LIN {X 0,Y 514.688,Z 526.81,A -85,B 0,C 180,E1 4924.755,E2 4924.755} C_VEL
LIN {X 0,Y 514.758,Z 527.266,A -85,B 0,C 180,E1 4925.27,E2 4925.27} C_VEL
LIN {X 0,Y 521.785,Z 550.887,A -85,B 0,C 180,E1 4925.881,E2 4925.881} C_VEL
LIN {X 0,Y 521.448,Z 608.09,A -85,B 0,C 180,E1 4926.837,E2 4926.837} C_VEL
LIN {X 0,Y 520.391,Z 641.868,A -85,B 0,C 180,E1 4928.058,E2 4928.058} C_VEL
LIN {X 0,Y 519.091,Z 674.479,A -85,B 0,C 180,E1 4929.962,E2 4929.962} C_VEL
LIN {X 0,Y 517.777,Z 702.458,A -85,B 0,C 180,E1 4932.319,E2 4932.319} C_VEL
LIN {X 0,Y 516.718,Z 728.108,A -85,B 0,C 180,E1 4935.321,E2 4935.321} C_VEL
LIN {X 0,Y 516.002,Z 747.013,A -85,B 0,C 180,E1 4938.414,E2 4938.414} C_VEL
LIN {X 0,Y 515.59,Z 761.456,A -85,B 0,C 180,E1 4941.986,E2 4941.986} C_VEL
LIN {X 0,Y 515.379,Z 770.612,A -85,B 0,C 180,E1 4945.792,E2 4945.792} C_VEL
LIN {X 0,Y 515.287,Z 773.417,A -85,B 0,C 180,E1 4948.32,E2 4948.32} C_VEL
LIN {X 0,Y 515.26,Z 773.413,A -85,B 0,C 180,E1 4951.688,E2 4951.688} C_VEL
LIN {X 0,Y 515.437,Z 769.059,A -85,B 0,C 180,E1 4955.06,E2 4955.06} C_VEL
LIN {X 0,Y 515.609,Z 758.543,A -85,B 0,C 180,E1 4958.872,E2 4958.872} C_VEL
LIN {X 0,Y 516.12,Z 743.377,A -85,B 0,C 180,E1 4962.284,E2 4962.284} C_VEL
LIN {X 0,Y 516.954,Z 721.721,A -85,B 0,C 180,E1 4965.505,E2 4965.505} C_VEL
LIN {X 0,Y 518.045,Z 696.57,A -85,B 0,C 180,E1 4968.199,E2 4968.199} C_VEL
LIN {X 0,Y 519.285,Z 666.936,A -85,B 0,C 180,E1 4970.484,E2 4970.484} C_VEL
LIN {X 0,Y 520.508,Z 633.588,A -85,B 0,C 180,E1 4972.223,E2 4972.223} C_VEL
LIN {X 0,Y 521.281,Z 599.339,A -85,B 0,C 180,E1 4973.289,E2 4973.289} C_VEL
LIN {X 0,Y 520.882,Z 547.826,A -85,B 0,C 180,E1 4974.084,E2 4974.084} C_VEL
LIN {X 0,Y 514.768,Z 526.81,A -85,B 0,C 180,E1 4974.643,E2 4974.643} C_VEL
LIN {X 0,Y 514.416,Z 526.81,A -85,B 0,C 180,E1 4980.028,E2 4980.028} C_VEL
LIN {X 0,Y 514.392,Z 526.81,A -85,B 0,C 180,E1 4986.068,E2 4986.068} C_VEL
LIN {X 0,Y 514.463,Z 526.81,A -85,B 0,C 180,E1 4990.356,E2 4990.356} C_VEL
LIN {X 0,Y 514.437,Z 526.81,A -85,B 0,C 180,E1 4995.071,E2 4995.071} C_VEL
LIN {X 0,Y 514.39,Z 526.81,A -85,B 0,C 180,E1 4999.939,E2 4999.939} C_VEL
LIN {X 0,Y 514.441,Z 526.81,A -85,B 0,C 180,E1 5006.008,E2 5006.008} C_VEL
LIN {X 0,Y 514.47,Z 526.81,A -85,B 0,C 180,E1 5012.001,E2 5012.001} C_VEL
LIN {X 0,Y 514.564,Z 526.81,A -85,B 0,C 180,E1 5017.517,E2 5017.517} C_VEL
LIN {X 0,Y 514.664,Z 526.81,A -85,B 0,C 180,E1 5022.898,E2 5022.898} C_VEL
LIN {X 0,Y 514.737,Z 526.81,A -85,B 0,C 180,E1 5025.56,E2 5025.56} C_VEL
LIN {X 0,Y 517.998,Z 546.221,A -85,B 0,C 180,E1 5026.403,E2 5026.403} C_VEL
LIN {X 0,Y 517.334,Z 571.62,A -85,B 0,C 180,E1 5027.97,E2 5027.97} C_VEL
LIN {X 0,Y 516.727,Z 591.359,A -85,B 0,C 180,E1 5029.88,E2 5029.88} C_VEL
LIN {X 0,Y 516.135,Z 608.515,A -85,B 0,C 180,E1 5032.42,E2 5032.42} C_VEL
LIN {X 0,Y 515.867,Z 619.171,A -85,B 0,C 180,E1 5034.954,E2 5034.954} C_VEL
LIN {X 0,Y 515.691,Z 625.064,A -85,B 0,C 180,E1 5037.487,E2 5037.487} C_VEL
LIN {X 0,Y 515.608,Z 626.839,A -85,B 0,C 180,E1 5040.005,E2 5040.005} C_VEL
LIN {X 0,Y 515.629,Z 623.406,A -85,B 0,C 180,E1 5043.213,E2 5043.213} C_VEL
LIN {X 0,Y 515.852,Z 615.231,A -85,B 0,C 180,E1 5045.901,E2 5045.901} C_VEL
LIN {X 0,Y 516.222,Z 600.778,A -85,B 0,C 180,E1 5048.65,E2 5048.65} C_VEL
LIN {X 0,Y 516.872,Z 581.15,A -85,B 0,C 180,E1 5051.001,E2 5051.001} C_VEL
LIN {X 0,Y 517.528,Z 557.908,A -85,B 0,C 180,E1 5052.787,E2 5052.787} C_VEL
LIN {X 0,Y 517.046,Z 538.572,A -85,B 0,C 180,E1 5053.772,E2 5053.772} C_VEL
LIN {X 0,Y 514.697,Z 526.81,A -85,B 0,C 180,E1 5054.253,E2 5054.253} C_VEL
LIN {X 0,Y 514.685,Z 526.81,A -85,B 0,C 180,E1 5060.676,E2 5060.676} C_VEL
LIN {X 0,Y 514.527,Z 526.81,A -85,B 0,C 180,E1 5066.197,E2 5066.197} C_VEL
LIN {X 0,Y 514.451,Z 526.81,A -85,B 0,C 180,E1 5071.993,E2 5071.993} C_VEL
LIN {X 0,Y 514.35,Z 526.81,A -85,B 0,C 180,E1 5078.187,E2 5078.187} C_VEL
LIN {X 0,Y 514.383,Z 526.81,A -85,B 0,C 180,E1 5082.614,E2 5082.614} C_VEL
LIN {X 0,Y 514.454,Z 526.81,A -85,B 0,C 180,E1 5087.393,E2 5087.393} C_VEL
LIN {X 0,Y 514.418,Z 526.81,A -85,B 0,C 180,E1 5092.63,E2 5092.63} C_VEL
LIN {X 0,Y 514.465,Z 526.81,A -85,B 0,C 180,E1 5098.596,E2 5098.596} C_VEL
LIN {X 0,Y 514.59,Z 526.81,A -85,B 0,C 180,E1 5103.806,E2 5103.806} C_VEL
LIN {X 0,Y 514.732,Z 526.81,A -85,B 0,C 180,E1 5110.273,E2 5110.273} C_VEL
LIN {X 0,Y 514.556,Z 526.81,A -85,B 0,C 180,E1 5116.182,E2 5116.182} C_VEL
LIN {X 0,Y 514.81,Z 526.81,A -85,B 0,C 180,E1 5121.54,E2 5121.54} C_VEL
LIN {X 0,Y 514.937,Z 526.81,A -85,B 0,C 180,E1 5126.625,E2 5126.625} C_VEL
LIN {X 0,Y 514.987,Z 526.81,A -85,B 0,C 180,E1 5131.681,E2 5131.681} C_VEL
LIN {X 0,Y 514.883,Z 526.81,A -85,B 0,C 180,E1 5136.751,E2 5136.751} C_VEL
LIN {X 0,Y 514.793,Z 526.81,A -85,B 0,C 180,E1 5141.877,E2 5141.877} C_VEL
LIN {X 0,Y 514.743,Z 526.81,A -85,B 0,C 180,E1 5147.102,E2 5147.102} C_VEL
LIN {X 0,Y 514.65,Z 526.81,A -85,B 0,C 180,E1 5152.481,E2 5152.481} C_VEL
LIN {X 0,Y 514.451,Z 526.81,A -85,B 0,C 180,E1 5158.088,E2 5158.088} C_VEL
LIN {X 0,Y 514.406,Z 526.81,A -85,B 0,C 180,E1 5163.998,E2 5163.998} C_VEL
LIN {X 0,Y 514.349,Z 526.81,A -85,B 0,C 180,E1 5170.356,E2 5170.356} C_VEL
LIN {X 0,Y 514.362,Z 526.81,A -85,B 0,C 180,E1 5175.048,E2 5175.048} C_VEL
LIN {X 0,Y 514.463,Z 526.81,A -85,B 0,C 180,E1 5179.917,E2 5179.917} C_VEL
LIN {X 0,Y 514.391,Z 526.81,A -85,B 0,C 180,E1 5185.992,E2 5185.992} C_VEL
LIN {X 0,Y 514.506,Z 526.81,A -85,B 0,C 180,E1 5191.977,E2 5191.977} C_VEL
LIN {X 0,Y 514.644,Z 526.81,A -85,B 0,C 180,E1 5197.51,E2 5197.51} C_VEL
LIN {X 0,Y 514.782,Z 526.81,A -85,B 0,C 180,E1 5202.891,E2 5202.891} C_VEL
LIN {X 0,Y 514.841,Z 526.81,A -85,B 0,C 180,E1 5209.832,E2 5209.832} C_VEL
LIN {X 0,Y 514.957,Z 526.81,A -85,B 0,C 180,E1 5214.935,E2 5214.935} C_VEL
LIN {X 0,Y 515.018,Z 526.81,A -85,B 0,C 180,E1 5219.995,E2 5219.995} C_VEL
LIN {X 0,Y 514.941,Z 526.81,A -85,B 0,C 180,E1 5225.055,E2 5225.055} C_VEL
LIN {X 0,Y 514.829,Z 526.81,A -85,B 0,C 180,E1 5230.158,E2 5230.158} C_VEL
LIN {X 0,Y 514.743,Z 526.81,A -85,B 0,C 180,E1 5235.344,E2 5235.344} C_VEL
LIN {X 0,Y 514.647,Z 526.81,A -85,B 0,C 180,E1 5240.666,E2 5240.666} C_VEL
LIN {X 0,Y 514.531,Z 526.81,A -85,B 0,C 180,E1 5246.186,E2 5246.186} C_VEL
LIN {X 0,Y 514.528,Z 526.81,A -85,B 0,C 180,E1 5251.975,E2 5251.975} C_VEL
LIN {X 0,Y 514.451,Z 526.81,A -85,B 0,C 180,E1 5256.471,E2 5256.471} C_VEL
LIN {X 0,Y 511.842,Z 526.81,A -85,B 0,C 180,E1 5257.91,E2 5257.91} C_VEL
LIN {X 0,Y 506.421,Z 526.81,A -85,B 0,C 180,E1 5260.067,E2 5260.067} C_VEL
LIN {X 0,Y 506.328,Z 526.81,A -85,B 0,C 180,E1 5260.317,E2 5260.317} C_VEL
LIN {X 0,Y 506.253,Z 526.81,A -85,B 0,C 180,E1 5266.544,E2 5266.544} C_VEL
LIN {X 0,Y 506.403,Z 526.81,A -85,B 0,C 180,E1 5273.28,E2 5273.28} C_VEL
LIN {X 0,Y 506.548,Z 526.81,A -85,B 0,C 180,E1 5280.074,E2 5280.074} C_VEL
LIN {X 0,Y 506.848,Z 527.611,A -85,B 0,C 180,E1 5284.953,E2 5284.953} C_VEL
LIN {X 0,Y 514.324,Z 552.741,A -85,B 0,C 180,E1 5285.621,E2 5285.621} C_VEL
LIN {X 0,Y 513.938,Z 607.892,A -85,B 0,C 180,E1 5286.567,E2 5286.567} C_VEL
LIN {X 0,Y 512.808,Z 641.417,A -85,B 0,C 180,E1 5287.803,E2 5287.803} C_VEL
LIN {X 0,Y 511.466,Z 672.724,A -85,B 0,C 180,E1 5289.65,E2 5289.65} C_VEL
LIN {X 0,Y 510.038,Z 700.829,A -85,B 0,C 180,E1 5292.025,E2 5292.025} C_VEL
LIN {X 0,Y 508.944,Z 725.749,A -85,B 0,C 180,E1 5294.937,E2 5294.937} C_VEL
LIN {X 0,Y 508.148,Z 745.662,A -85,B 0,C 180,E1 5298.184,E2 5298.184} C_VEL
LIN {X 0,Y 507.69,Z 761.118,A -85,B 0,C 180,E1 5301.86,E2 5301.86} C_VEL
LIN {X 0,Y 507.531,Z 769.038,A -85,B 0,C 180,E1 5304.869,E2 5304.869} C_VEL
LIN {X 0,Y 507.402,Z 773.417,A -85,B 0,C 180,E1 5308.294,E2 5308.294} C_VEL
LIN {X 0,Y 507.377,Z 773.412,A -85,B 0,C 180,E1 5311.714,E2 5311.714} C_VEL
LIN {X 0,Y 507.536,Z 769.022,A -85,B 0,C 180,E1 5315.139,E2 5315.139} C_VEL
LIN {X 0,Y 507.699,Z 759.639,A -85,B 0,C 180,E1 5318.579,E2 5318.579} C_VEL
LIN {X 0,Y 508.191,Z 744.342,A -85,B 0,C 180,E1 5322.042,E2 5322.042} C_VEL
LIN {X 0,Y 509.032,Z 722.96,A -85,B 0,C 180,E1 5325.379,E2 5325.379} C_VEL
LIN {X 0,Y 510.201,Z 696.837,A -85,B 0,C 180,E1 5328.289,E2 5328.289} C_VEL
LIN {X 0,Y 511.579,Z 666.289,A -85,B 0,C 180,E1 5330.694,E2 5330.694} C_VEL
LIN {X 0,Y 512.856,Z 633.34,A -85,B 0,C 180,E1 5332.445,E2 5332.445} C_VEL
LIN {X 0,Y 513.719,Z 598.789,A -85,B 0,C 180,E1 5333.543,E2 5333.543} C_VEL
LIN {X 0,Y 513.227,Z 549.236,A -85,B 0,C 180,E1 5334.327,E2 5334.327} C_VEL
LIN {X 0,Y 506.836,Z 526.81,A -85,B 0,C 180,E1 5334.925,E2 5334.925} C_VEL
LIN {X 0,Y 506.487,Z 526.81,A -85,B 0,C 180,E1 5340.548,E2 5340.548} C_VEL
LIN {X 0,Y 506.494,Z 526.81,A -85,B 0,C 180,E1 5346.722,E2 5346.722} C_VEL
LIN {X 0,Y 506.5,Z 526.81,A -85,B 0,C 180,E1 5353.441,E2 5353.441} C_VEL
LIN {X 0,Y 506.41,Z 526.81,A -85,B 0,C 180,E1 5358.881,E2 5358.881} C_VEL
LIN {X 0,Y 506.509,Z 526.81,A -85,B 0,C 180,E1 5365.401,E2 5365.401} C_VEL
LIN {X 0,Y 506.516,Z 526.81,A -85,B 0,C 180,E1 5371.435,E2 5371.435} C_VEL
LIN {X 0,Y 506.655,Z 526.81,A -85,B 0,C 180,E1 5377.89,E2 5377.89} C_VEL
LIN {X 0,Y 506.771,Z 526.81,A -85,B 0,C 180,E1 5382.965,E2 5382.965} C_VEL
LIN {X 0,Y 506.844,Z 527.591,A -85,B 0,C 180,E1 5385.305,E2 5385.305} C_VEL
LIN {X 0,Y 510.386,Z 547.579,A -85,B 0,C 180,E1 5386.203,E2 5386.203} C_VEL
LIN {X 0,Y 509.691,Z 572.731,A -85,B 0,C 180,E1 5387.787,E2 5387.787} C_VEL
LIN {X 0,Y 509.05,Z 592.486,A -85,B 0,C 180,E1 5389.726,E2 5389.726} C_VEL
LIN {X 0,Y 508.39,Z 609.683,A -85,B 0,C 180,E1 5392.304,E2 5392.304} C_VEL
LIN {X 0,Y 508.1,Z 620.358,A -85,B 0,C 180,E1 5394.877,E2 5394.877} C_VEL
LIN {X 0,Y 507.914,Z 626.246,A -85,B 0,C 180,E1 5397.448,E2 5397.448} C_VEL
LIN {X 0,Y 507.823,Z 627.99,A -85,B 0,C 180,E1 5400.005,E2 5400.005} C_VEL
LIN {X 0,Y 507.843,Z 625.868,A -85,B 0,C 180,E1 5402.499,E2 5402.499} C_VEL
LIN {X 0,Y 508.042,Z 617.866,A -85,B 0,C 180,E1 5405.563,E2 5405.563} C_VEL
LIN {X 0,Y 508.348,Z 604.4,A -85,B 0,C 180,E1 5408.354,E2 5408.354} C_VEL
LIN {X 0,Y 508.997,Z 586.155,A -85,B 0,C 180,E1 5410.743,E2 5410.743} C_VEL
LIN {X 0,Y 509.741,Z 563.664,A -85,B 0,C 180,E1 5412.658,E2 5412.658} C_VEL
LIN {X 0,Y 509.573,Z 540.716,A -85,B 0,C 180,E1 5413.922,E2 5413.922} C_VEL
LIN {X 0,Y 506.772,Z 526.81,A -85,B 0,C 180,E1 5414.533,E2 5414.533} C_VEL
LIN {X 0,Y 506.737,Z 526.81,A -85,B 0,C 180,E1 5421.015,E2 5421.015} C_VEL
LIN {X 0,Y 506.603,Z 526.81,A -85,B 0,C 180,E1 5426.639,E2 5426.639} C_VEL
LIN {X 0,Y 506.475,Z 526.81,A -85,B 0,C 180,E1 5432.559,E2 5432.559} C_VEL
LIN {X 0,Y 506.436,Z 526.81,A -85,B 0,C 180,E1 5436.726,E2 5436.726} C_VEL
LIN {X 0,Y 506.391,Z 526.81,A -85,B 0,C 180,E1 5443.451,E2 5443.451} C_VEL
LIN {X 0,Y 506.469,Z 526.81,A -85,B 0,C 180,E1 5448.871,E2 5448.871} C_VEL
LIN {X 0,Y 506.491,Z 526.81,A -85,B 0,C 180,E1 5455.386,E2 5455.386} C_VEL
LIN {X 0,Y 506.565,Z 526.81,A -85,B 0,C 180,E1 5461.426,E2 5461.426} C_VEL
LIN {X 0,Y 506.761,Z 526.81,A -85,B 0,C 180,E1 5467.856,E2 5467.856} C_VEL
LIN {X 0,Y 506.849,Z 526.81,A -85,B 0,C 180,E1 5472.931,E2 5472.931} C_VEL
LIN {X 0,Y 506.89,Z 526.81,A -85,B 0,C 180,E1 5479.672,E2 5479.672} C_VEL
LIN {X 0,Y 507.082,Z 526.81,A -85,B 0,C 180,E1 5484.857,E2 5484.857} C_VEL
LIN {X 0,Y 507.175,Z 526.81,A -85,B 0,C 180,E1 5489.996,E2 5489.996} C_VEL
LIN {X 0,Y 507.057,Z 526.81,A -85,B 0,C 180,E1 5495.135,E2 5495.135} C_VEL
LIN {X 0,Y 506.959,Z 526.81,A -85,B 0,C 180,E1 5500.319,E2 5500.319} C_VEL
LIN {X 0,Y 506.85,Z 526.81,A -85,B 0,C 180,E1 5505.592,E2 5505.592} C_VEL
LIN {X 0,Y 506.742,Z 526.81,A -85,B 0,C 180,E1 5511.006,E2 5511.006} C_VEL
LIN {X 0,Y 506.587,Z 526.81,A -85,B 0,C 180,E1 5516.631,E2 5516.631} C_VEL
LIN {X 0,Y 506.466,Z 526.81,A -85,B 0,C 180,E1 5522.55,E2 5522.55} C_VEL
LIN {X 0,Y 506.459,Z 526.81,A -85,B 0,C 180,E1 5526.715,E2 5526.715} C_VEL
LIN {X 0,Y 506.345,Z 526.81,A -85,B 0,C 180,E1 5533.446,E2 5533.446} C_VEL
LIN {X 0,Y 506.463,Z 526.81,A -85,B 0,C 180,E1 5538.872,E2 5538.872} C_VEL
LIN {X 0,Y 506.477,Z 526.81,A -85,B 0,C 180,E1 5545.386,E2 5545.386} C_VEL
LIN {X 0,Y 506.532,Z 526.81,A -85,B 0,C 180,E1 5551.424,E2 5551.424} C_VEL
LIN {X 0,Y 506.746,Z 526.81,A -85,B 0,C 180,E1 5557.843,E2 5557.843} C_VEL
LIN {X 0,Y 506.898,Z 526.81,A -85,B 0,C 180,E1 5562.891,E2 5562.891} C_VEL
LIN {X 0,Y 506.91,Z 526.81,A -85,B 0,C 180,E1 5569.671,E2 5569.671} C_VEL
LIN {X 0,Y 507.05,Z 526.81,A -85,B 0,C 180,E1 5574.855,E2 5574.855} C_VEL
LIN {X 0,Y 507.137,Z 526.81,A -85,B 0,C 180,E1 5579.995,E2 5579.995} C_VEL
LIN {X 0,Y 507.026,Z 526.81,A -85,B 0,C 180,E1 5585.134,E2 5585.134} C_VEL
LIN {X 0,Y 506.901,Z 526.81,A -85,B 0,C 180,E1 5590.318,E2 5590.318} C_VEL
LIN {X 0,Y 506.81,Z 526.81,A -85,B 0,C 180,E1 5595.591,E2 5595.591} C_VEL
LIN {X 0,Y 506.699,Z 526.81,A -85,B 0,C 180,E1 5601.006,E2 5601.006} C_VEL
LIN {X 0,Y 506.589,Z 526.81,A -85,B 0,C 180,E1 5606.628,E2 5606.628} C_VEL
LIN {X 0,Y 506.554,Z 526.81,A -85,B 0,C 180,E1 5612.54,E2 5612.54} C_VEL
LIN {X 0,Y 506.552,Z 526.81,A -85,B 0,C 180,E1 5616.703,E2 5616.703} C_VEL
LIN {X 0,Y 506.328,Z 526.81,A -85,B 0,C 180,E1 5620.317,E2 5620.317} C_VEL
LIN {X 0,Y 503.776,Z 526.81,A -85,B 0,C 180,E1 5621.776,E2 5621.776} C_VEL
LIN {X 0,Y 498.424,Z 526.81,A -85,B 0,C 180,E1 5623.964,E2 5623.964} C_VEL
LIN {X 0,Y 498.34,Z 526.81,A -85,B 0,C 180,E1 5624.217,E2 5624.217} C_VEL
LIN {X 0,Y 498.353,Z 526.81,A -85,B 0,C 180,E1 5630.362,E2 5630.362} C_VEL
LIN {X 0,Y 498.519,Z 526.81,A -85,B 0,C 180,E1 5636.865,E2 5636.865} C_VEL
LIN {X 0,Y 498.674,Z 526.81,A -85,B 0,C 180,E1 5642.912,E2 5642.912} C_VEL
LIN {X 0,Y 498.945,Z 527.599,A -85,B 0,C 180,E1 5644.618,E2 5644.618} C_VEL
LIN {X 0,Y 506.883,Z 555.382,A -85,B 0,C 180,E1 5645.365,E2 5645.365} C_VEL
LIN {X 0,Y 506.433,Z 607.155,A -85,B 0,C 180,E1 5646.274,E2 5646.274} C_VEL
LIN {X 0,Y 505.289,Z 639.839,A -85,B 0,C 180,E1 5647.484,E2 5647.484} C_VEL
LIN {X 0,Y 503.819,Z 670.962,A -85,B 0,C 180,E1 5649.327,E2 5649.327} C_VEL
LIN {X 0,Y 502.324,Z 699.692,A -85,B 0,C 180,E1 5651.773,E2 5651.773} C_VEL
LIN {X 0,Y 501.089,Z 725.23,A -85,B 0,C 180,E1 5654.81,E2 5654.81} C_VEL
LIN {X 0,Y 500.269,Z 745.59,A -85,B 0,C 180,E1 5658.216,E2 5658.216} C_VEL
LIN {X 0,Y 499.821,Z 759.982,A -85,B 0,C 180,E1 5661.731,E2 5661.731} C_VEL
LIN {X 0,Y 499.686,Z 768.054,A -85,B 0,C 180,E1 5664.789,E2 5664.789} C_VEL
LIN {X 0,Y 499.554,Z 772.641,A -85,B 0,C 180,E1 5668.267,E2 5668.267} C_VEL
LIN {X 0,Y 499.511,Z 772.62,A -85,B 0,C 180,E1 5671.741,E2 5671.741} C_VEL
LIN {X 0,Y 499.692,Z 767.992,A -85,B 0,C 180,E1 5675.22,E2 5675.22} C_VEL
LIN {X 0,Y 499.843,Z 758.366,A -85,B 0,C 180,E1 5678.715,E2 5678.715} C_VEL
LIN {X 0,Y 500.378,Z 741.785,A -85,B 0,C 180,E1 5682.454,E2 5682.454} C_VEL
LIN {X 0,Y 501.283,Z 720.185,A -85,B 0,C 180,E1 5685.778,E2 5685.778} C_VEL
LIN {X 0,Y 502.447,Z 694.917,A -85,B 0,C 180,E1 5688.581,E2 5688.581} C_VEL
LIN {X 0,Y 503.852,Z 665.634,A -85,B 0,C 180,E1 5690.911,E2 5690.911} C_VEL
LIN {X 0,Y 505.281,Z 632.443,A -85,B 0,C 180,E1 5692.701,E2 5692.701} C_VEL
LIN {X 0,Y 506.145,Z 597.687,A -85,B 0,C 180,E1 5693.817,E2 5693.817} C_VEL
LIN {X 0,Y 505.55,Z 550.499,A -85,B 0,C 180,E1 5694.582,E2 5694.582} C_VEL
LIN {X 0,Y 498.916,Z 526.81,A -85,B 0,C 180,E1 5695.242,E2 5695.242} C_VEL
LIN {X 0,Y 498.5,Z 526.81,A -85,B 0,C 180,E1 5701.757,E2 5701.757} C_VEL
LIN {X 0,Y 498.504,Z 526.81,A -85,B 0,C 180,E1 5707.857,E2 5707.857} C_VEL
LIN {X 0,Y 498.576,Z 526.81,A -85,B 0,C 180,E1 5714.309,E2 5714.309} C_VEL
LIN {X 0,Y 498.443,Z 526.81,A -85,B 0,C 180,E1 5720.374,E2 5720.374} C_VEL
LIN {X 0,Y 498.633,Z 526.81,A -85,B 0,C 180,E1 5726.877,E2 5726.877} C_VEL
LIN {X 0,Y 498.606,Z 526.81,A -85,B 0,C 180,E1 5732.911,E2 5732.911} C_VEL
LIN {X 0,Y 498.755,Z 526.81,A -85,B 0,C 180,E1 5738.643,E2 5738.643} C_VEL
LIN {X 0,Y 498.867,Z 526.988,A -85,B 0,C 180,E1 5744.99,E2 5744.99} C_VEL
LIN {X 0,Y 502.812,Z 548.43,A -85,B 0,C 180,E1 5745.968,E2 5745.968} C_VEL
LIN {X 0,Y 502.08,Z 573.876,A -85,B 0,C 180,E1 5747.599,E2 5747.599} C_VEL
LIN {X 0,Y 501.358,Z 593.615,A -85,B 0,C 180,E1 5749.567,E2 5749.567} C_VEL
LIN {X 0,Y 500.648,Z 610.846,A -85,B 0,C 180,E1 5752.184,E2 5752.184} C_VEL
LIN {X 0,Y 500.338,Z 621.541,A -85,B 0,C 180,E1 5754.797,E2 5754.797} C_VEL
LIN {X 0,Y 500.072,Z 627.84,A -85,B 0,C 180,E1 5757.725,E2 5757.725} C_VEL
LIN {X 0,Y 500.009,Z 629.144,A -85,B 0,C 180,E1 5760.005,E2 5760.005} C_VEL
LIN {X 0,Y 500.035,Z 626.869,A -85,B 0,C 180,E1 5762.608,E2 5762.608} C_VEL
LIN {X 0,Y 500.242,Z 618.882,A -85,B 0,C 180,E1 5765.65,E2 5765.65} C_VEL
LIN {X 0,Y 500.585,Z 605.307,A -85,B 0,C 180,E1 5768.484,E2 5768.484} C_VEL
LIN {X 0,Y 501.296,Z 586.962,A -85,B 0,C 180,E1 5770.91,E2 5770.91} C_VEL
LIN {X 0,Y 502.091,Z 564.389,A -85,B 0,C 180,E1 5772.855,E2 5772.855} C_VEL
LIN {X 0,Y 501.919,Z 541.672,A -85,B 0,C 180,E1 5774.129,E2 5774.129} C_VEL
LIN {X 0,Y 498.87,Z 526.81,A -85,B 0,C 180,E1 5774.844,E2 5774.844} C_VEL
LIN {X 0,Y 498.833,Z 526.81,A -85,B 0,C 180,E1 5781.365,E2 5781.365} C_VEL
LIN {X 0,Y 498.631,Z 526.81,A -85,B 0,C 180,E1 5787.1,E2 5787.1} C_VEL
LIN {X 0,Y 498.563,Z 526.81,A -85,B 0,C 180,E1 5793.141,E2 5793.141} C_VEL
LIN {X 0,Y 498.435,Z 526.81,A -85,B 0,C 180,E1 5799.64,E2 5799.64} C_VEL
LIN {X 0,Y 498.544,Z 526.81,A -85,B 0,C 180,E1 5805.687,E2 5805.687} C_VEL
LIN {X 0,Y 498.516,Z 526.81,A -85,B 0,C 180,E1 5812.159,E2 5812.159} C_VEL
LIN {X 0,Y 498.538,Z 526.81,A -85,B 0,C 180,E1 5818.257,E2 5818.257} C_VEL
LIN {X 0,Y 498.677,Z 526.81,A -85,B 0,C 180,E1 5822.903,E2 5822.903} C_VEL
LIN {X 0,Y 498.859,Z 526.81,A -85,B 0,C 180,E1 5828.637,E2 5828.637} C_VEL
LIN {X 0,Y 498.829,Z 526.81,A -85,B 0,C 180,E1 5834.143,E2 5834.143} C_VEL
LIN {X 0,Y 498.956,Z 526.81,A -85,B 0,C 180,E1 5839.506,E2 5839.506} C_VEL
LIN {X 0,Y 499.192,Z 526.81,A -85,B 0,C 180,E1 5844.775,E2 5844.775} C_VEL
LIN {X 0,Y 499.299,Z 526.81,A -85,B 0,C 180,E1 5849.996,E2 5849.996} C_VEL
LIN {X 0,Y 499.164,Z 526.81,A -85,B 0,C 180,E1 5855.217,E2 5855.217} C_VEL
LIN {X 0,Y 499.03,Z 526.81,A -85,B 0,C 180,E1 5860.484,E2 5860.484} C_VEL
LIN {X 0,Y 498.937,Z 526.81,A -85,B 0,C 180,E1 5865.845,E2 5865.845} C_VEL
LIN {X 0,Y 498.833,Z 526.81,A -85,B 0,C 180,E1 5871.356,E2 5871.356} C_VEL
LIN {X 0,Y 498.612,Z 526.81,A -85,B 0,C 180,E1 5877.091,E2 5877.091} C_VEL
LIN {X 0,Y 498.557,Z 526.81,A -85,B 0,C 180,E1 5883.132,E2 5883.132} C_VEL
LIN {X 0,Y 498.411,Z 526.81,A -85,B 0,C 180,E1 5889.633,E2 5889.633} C_VEL
LIN {X 0,Y 498.509,Z 526.81,A -85,B 0,C 180,E1 5895.684,E2 5895.684} C_VEL
LIN {X 0,Y 498.497,Z 526.81,A -85,B 0,C 180,E1 5902.15,E2 5902.15} C_VEL
LIN {X 0,Y 498.557,Z 526.81,A -85,B 0,C 180,E1 5908.24,E2 5908.24} C_VEL
LIN {X 0,Y 498.741,Z 526.81,A -85,B 0,C 180,E1 5914.844,E2 5914.844} C_VEL
LIN {X 0,Y 498.952,Z 526.81,A -85,B 0,C 180,E1 5920.496,E2 5920.496} C_VEL
LIN {X 0,Y 498.79,Z 526.81,A -85,B 0,C 180,E1 5926.235,E2 5926.235} C_VEL
LIN {X 0,Y 499.005,Z 526.81,A -85,B 0,C 180,E1 5931.393,E2 5931.393} C_VEL
LIN {X 0,Y 499.12,Z 526.81,A -85,B 0,C 180,E1 5936.517,E2 5936.517} C_VEL
LIN {X 0,Y 499.197,Z 526.81,A -85,B 0,C 180,E1 5941.733,E2 5941.733} C_VEL
LIN {X 0,Y 499.022,Z 526.81,A -85,B 0,C 180,E1 5946.965,E2 5946.965} C_VEL
LIN {X 0,Y 498.903,Z 526.81,A -85,B 0,C 180,E1 5952.259,E2 5952.259} C_VEL
LIN {X 0,Y 498.851,Z 526.81,A -85,B 0,C 180,E1 5957.662,E2 5957.662} C_VEL
LIN {X 0,Y 498.723,Z 526.81,A -85,B 0,C 180,E1 5963.238,E2 5963.238} C_VEL
LIN {X 0,Y 498.633,Z 526.81,A -85,B 0,C 180,E1 5969.059,E2 5969.059} C_VEL
LIN {X 0,Y 498.637,Z 526.81,A -85,B 0,C 180,E1 5975.225,E2 5975.225} C_VEL
LIN {X 0,Y 498.425,Z 526.81,A -85,B 0,C 180,E1 5981.926,E2 5981.926} C_VEL
LIN {X 0,Y 498.34,Z 526.81,A -85,B 0,C 180,E1 5984.217,E2 5984.217} C_VEL
LIN {X 0,Y 495.868,Z 526.81,A -85,B 0,C 180,E1 5985.694,E2 5985.694} C_VEL
LIN {X 0,Y 490.389,Z 526.81,A -85,B 0,C 180,E1 5988.164,E2 5988.164} C_VEL
LIN {X 0,Y 490.482,Z 526.81,A -85,B 0,C 180,E1 5994.095,E2 5994.095} C_VEL
LIN {X 0,Y 490.623,Z 526.81,A -85,B 0,C 180,E1 6000.417,E2 6000.417} C_VEL
LIN {X 0,Y 490.974,Z 526.81,A -85,B 0,C 180,E1 6004.243,E2 6004.243} C_VEL
LIN {X 0,Y 499.458,Z 557.084,A -85,B 0,C 180,E1 6005.088,E2 6005.088} C_VEL
LIN {X 0,Y 498.938,Z 606.435,A -85,B 0,C 180,E1 6005.972,E2 6005.972} C_VEL
LIN {X 0,Y 497.685,Z 639.961,A -85,B 0,C 180,E1 6007.241,E2 6007.241} C_VEL
LIN {X 0,Y 496.111,Z 670.795,A -85,B 0,C 180,E1 6009.108,E2 6009.108} C_VEL
LIN {X 0,Y 494.51,Z 699.615,A -85,B 0,C 180,E1 6011.622,E2 6011.622} C_VEL
LIN {X 0,Y 493.25,Z 723.446,A -85,B 0,C 180,E1 6014.493,E2 6014.493} C_VEL
LIN {X 0,Y 492.384,Z 744.374,A -85,B 0,C 180,E1 6018.025,E2 6018.025} C_VEL
LIN {X 0,Y 491.952,Z 758.846,A -85,B 0,C 180,E1 6021.598,E2 6021.598} C_VEL
LIN {X 0,Y 491.862,Z 766.957,A -85,B 0,C 180,E1 6024.706,E2 6024.706} C_VEL
LIN {X 0,Y 491.73,Z 771.546,A -85,B 0,C 180,E1 6028.24,E2 6028.24} C_VEL
LIN {X 0,Y 491.689,Z 771.501,A -85,B 0,C 180,E1 6031.769,E2 6031.769} C_VEL
LIN {X 0,Y 491.868,Z 766.82,A -85,B 0,C 180,E1 6035.303,E2 6035.303} C_VEL
LIN {X 0,Y 492.019,Z 755.902,A -85,B 0,C 180,E1 6039.176,E2 6039.176} C_VEL
LIN {X 0,Y 492.53,Z 740.378,A -85,B 0,C 180,E1 6042.656,E2 6042.656} C_VEL
LIN {X 0,Y 493.463,Z 718.565,A -85,B 0,C 180,E1 6046.034,E2 6046.034} C_VEL
LIN {X 0,Y 494.767,Z 692.021,A -85,B 0,C 180,E1 6048.973,E2 6048.973} C_VEL
LIN {X 0,Y 496.281,Z 661.539,A -85,B 0,C 180,E1 6051.362,E2 6051.362} C_VEL
LIN {X 0,Y 497.745,Z 629.42,A -85,B 0,C 180,E1 6053.061,E2 6053.061} C_VEL
LIN {X 0,Y 498.658,Z 594.607,A -85,B 0,C 180,E1 6054.143,E2 6054.143} C_VEL
LIN {X 0,Y 498.3,Z 552.911,A -85,B 0,C 180,E1 6054.817,E2 6054.817} C_VEL
LIN {X 0,Y 490.993,Z 526.81,A -85,B 0,C 180,E1 6055.581,E2 6055.581} C_VEL
LIN {X 0,Y 490.624,Z 526.81,A -85,B 0,C 180,E1 6061.648,E2 6061.648} C_VEL
LIN {X 0,Y 490.578,Z 526.81,A -85,B 0,C 180,E1 6068.122,E2 6068.122} C_VEL
LIN {X 0,Y 490.684,Z 526.81,A -85,B 0,C 180,E1 6072.759,E2 6072.759} C_VEL
LIN {X 0,Y 490.626,Z 526.81,A -85,B 0,C 180,E1 6077.792,E2 6077.792} C_VEL
LIN {X 0,Y 490.578,Z 526.81,A -85,B 0,C 180,E1 6084.107,E2 6084.107} C_VEL
LIN {X 0,Y 490.661,Z 526.81,A -85,B 0,C 180,E1 6090.422,E2 6090.422} C_VEL
LIN {X 0,Y 490.757,Z 526.81,A -85,B 0,C 180,E1 6096.362,E2 6096.362} C_VEL
LIN {X 0,Y 490.895,Z 526.81,A -85,B 0,C 180,E1 6102.042,E2 6102.042} C_VEL
LIN {X 0,Y 490.966,Z 527.217,A -85,B 0,C 180,E1 6104.683,E2 6104.683} C_VEL
LIN {X 0,Y 495.273,Z 549.769,A -85,B 0,C 180,E1 6105.75,E2 6105.75} C_VEL
LIN {X 0,Y 494.46,Z 575.07,A -85,B 0,C 180,E1 6107.405,E2 6107.405} C_VEL
LIN {X 0,Y 493.606,Z 596.531,A -85,B 0,C 180,E1 6109.624,E2 6109.624} C_VEL
LIN {X 0,Y 492.876,Z 613.122,A -85,B 0,C 180,E1 6112.282,E2 6112.282} C_VEL
LIN {X 0,Y 492.497,Z 624.019,A -85,B 0,C 180,E1 6115.156,E2 6115.156} C_VEL
LIN {X 0,Y 492.198,Z 629.608,A -85,B 0,C 180,E1 6118.243,E2 6118.243} C_VEL
LIN {X 0,Y 492.195,Z 630.299,A -85,B 0,C 180,E1 6120.005,E2 6120.005} C_VEL
LIN {X 0,Y 492.219,Z 627.966,A -85,B 0,C 180,E1 6122.65,E2 6122.65} C_VEL
LIN {X 0,Y 492.441,Z 619.885,A -85,B 0,C 180,E1 6125.74,E2 6125.74} C_VEL
LIN {X 0,Y 492.841,Z 606.211,A -85,B 0,C 180,E1 6128.618,E2 6128.618} C_VEL
LIN {X 0,Y 493.597,Z 588.033,A -85,B 0,C 180,E1 6131.053,E2 6131.053} C_VEL
LIN {X 0,Y 494.43,Z 565.108,A -85,B 0,C 180,E1 6133.057,E2 6133.057} C_VEL
LIN {X 0,Y 494.177,Z 542.399,A -85,B 0,C 180,E1 6134.355,E2 6134.355} C_VEL
LIN {X 0,Y 490.925,Z 526.81,A -85,B 0,C 180,E1 6135.092,E2 6135.092} C_VEL
LIN {X 0,Y 490.933,Z 526.81,A -85,B 0,C 180,E1 6139.836,E2 6139.836} C_VEL
LIN {X 0,Y 490.754,Z 526.81,A -85,B 0,C 180,E1 6145.594,E2 6145.594} C_VEL
LIN {X 0,Y 490.667,Z 526.81,A -85,B 0,C 180,E1 6151.644,E2 6151.644} C_VEL
LIN {X 0,Y 490.517,Z 526.81,A -85,B 0,C 180,E1 6158.126,E2 6158.126} C_VEL
LIN {X 0,Y 490.601,Z 526.81,A -85,B 0,C 180,E1 6164.774,E2 6164.774} C_VEL
LIN {X 0,Y 490.594,Z 526.81,A -85,B 0,C 180,E1 6170.498,E2 6170.498} C_VEL
LIN {X 0,Y 490.622,Z 526.81,A -85,B 0,C 180,E1 6176.437,E2 6176.437} C_VEL
LIN {X 0,Y 490.738,Z 526.81,A -85,B 0,C 180,E1 6182.428,E2 6182.428} C_VEL
LIN {X 0,Y 490.903,Z 526.81,A -85,B 0,C 180,E1 6188.273,E2 6188.273} C_VEL
LIN {X 0,Y 490.912,Z 526.81,A -85,B 0,C 180,E1 6193.88,E2 6193.88} C_VEL
LIN {X 0,Y 491.047,Z 526.81,A -85,B 0,C 180,E1 6200.65,E2 6200.65} C_VEL
LIN {X 0,Y 491.233,Z 526.81,A -85,B 0,C 180,E1 6206.462,E2 6206.462} C_VEL
LIN {X 0,Y 491.3,Z 526.81,A -85,B 0,C 180,E1 6211.762,E2 6211.762} C_VEL
LIN {X 0,Y 491.149,Z 526.81,A -85,B 0,C 180,E1 6217.079,E2 6217.079} C_VEL
LIN {X 0,Y 491.047,Z 526.81,A -85,B 0,C 180,E1 6222.46,E2 6222.46} C_VEL
LIN {X 0,Y 490.967,Z 526.81,A -85,B 0,C 180,E1 6227.957,E2 6227.957} C_VEL
LIN {X 0,Y 490.824,Z 526.81,A -85,B 0,C 180,E1 6233.637,E2 6233.637} C_VEL
LIN {X 0,Y 490.611,Z 526.81,A -85,B 0,C 180,E1 6240.214,E2 6240.214} C_VEL
LIN {X 0,Y 490.547,Z 526.81,A -85,B 0,C 180,E1 6245.899,E2 6245.899} C_VEL
LIN {X 0,Y 490.5,Z 526.81,A -85,B 0,C 180,E1 6252.193,E2 6252.193} C_VEL
LIN {X 0,Y 490.646,Z 526.81,A -85,B 0,C 180,E1 6257.777,E2 6257.777} C_VEL
LIN {X 0,Y 490.564,Z 526.81,A -85,B 0,C 180,E1 6264.093,E2 6264.093} C_VEL
LIN {X 0,Y 490.636,Z 526.81,A -85,B 0,C 180,E1 6270.408,E2 6270.408} C_VEL
LIN {X 0,Y 490.84,Z 526.81,A -85,B 0,C 180,E1 6276.354,E2 6276.354} C_VEL
LIN {X 0,Y 491.024,Z 526.81,A -85,B 0,C 180,E1 6282.035,E2 6282.035} C_VEL
LIN {X 0,Y 490.912,Z 526.81,A -85,B 0,C 180,E1 6287.527,E2 6287.527} C_VEL
LIN {X 0,Y 491.227,Z 526.81,A -85,B 0,C 180,E1 6292.913,E2 6292.913} C_VEL
LIN {X 0,Y 491.465,Z 526.81,A -85,B 0,C 180,E1 6298.229,E2 6298.229} C_VEL
LIN {X 0,Y 491.374,Z 526.81,A -85,B 0,C 180,E1 6303.528,E2 6303.528} C_VEL
LIN {X 0,Y 491.073,Z 526.81,A -85,B 0,C 180,E1 6309.41,E2 6309.41} C_VEL
LIN {X 0,Y 491.002,Z 526.81,A -85,B 0,C 180,E1 6314.275,E2 6314.275} C_VEL
LIN {X 0,Y 490.908,Z 526.81,A -85,B 0,C 180,E1 6319.825,E2 6319.825} C_VEL
LIN {X 0,Y 490.735,Z 526.81,A -85,B 0,C 180,E1 6325.583,E2 6325.583} C_VEL
LIN {X 0,Y 490.719,Z 526.81,A -85,B 0,C 180,E1 6331.628,E2 6331.628} C_VEL
LIN {X 0,Y 490.593,Z 526.81,A -85,B 0,C 180,E1 6338.106,E2 6338.106} C_VEL
LIN {X 0,Y 490.443,Z 526.81,A -85,B 0,C 180,E1 6344.768,E2 6344.768} C_VEL
LIN {X 0,Y 490.389,Z 526.81,A -85,B 0,C 180,E1 6348.164,E2 6348.164} C_VEL
LIN {X 0,Y 486.436,Z 526.81,A -85,B 0,C 180,E1 6350.15,E2 6350.15} C_VEL
LIN {X 0,Y 482.503,Z 526.81,A -85,B 0,C 180,E1 6352.168,E2 6352.168} C_VEL
LIN {X 0,Y 482.67,Z 526.81,A -85,B 0,C 180,E1 6357.867,E2 6357.867} C_VEL
LIN {X 0,Y 483.057,Z 527.203,A -85,B 0,C 180,E1 6363.916,E2 6363.916} C_VEL
LIN {X 0,Y 492.05,Z 558.866,A -85,B 0,C 180,E1 6364.806,E2 6364.806} C_VEL
LIN {X 0,Y 491.421,Z 607.293,A -85,B 0,C 180,E1 6365.706,E2 6365.706} C_VEL
LIN {X 0,Y 490.051,Z 641.141,A -85,B 0,C 180,E1 6367.046,E2 6367.046} C_VEL
LIN {X 0,Y 488.345,Z 672.811,A -85,B 0,C 180,E1 6369.045,E2 6369.045} C_VEL
LIN {X 0,Y 486.576,Z 702.077,A -85,B 0,C 180,E1 6371.734,E2 6371.734} C_VEL
LIN {X 0,Y 485.288,Z 725.925,A -85,B 0,C 180,E1 6374.805,E2 6374.805} C_VEL
LIN {X 0,Y 484.52,Z 745.343,A -85,B 0,C 180,E1 6378.285,E2 6378.285} C_VEL
LIN {X 0,Y 484.104,Z 759.126,A -85,B 0,C 180,E1 6381.914,E2 6381.914} C_VEL
LIN {X 0,Y 483.963,Z 767.487,A -85,B 0,C 180,E1 6385.518,E2 6385.518} C_VEL
LIN {X 0,Y 483.91,Z 770.45,A -85,B 0,C 180,E1 6388.211,E2 6388.211} C_VEL
LIN {X 0,Y 483.882,Z 770.384,A -85,B 0,C 180,E1 6391.797,E2 6391.797} C_VEL
LIN {X 0,Y 484.021,Z 765.645,A -85,B 0,C 180,E1 6395.389,E2 6395.389} C_VEL
LIN {X 0,Y 484.143,Z 755.814,A -85,B 0,C 180,E1 6399,E2 6399} C_VEL
LIN {X 0,Y 484.636,Z 740.122,A -85,B 0,C 180,E1 6402.636,E2 6402.636} C_VEL
LIN {X 0,Y 485.572,Z 718.746,A -85,B 0,C 180,E1 6406.059,E2 6406.059} C_VEL
LIN {X 0,Y 486.862,Z 693.21,A -85,B 0,C 180,E1 6408.993,E2 6408.993} C_VEL
LIN {X 0,Y 488.476,Z 663.19,A -85,B 0,C 180,E1 6411.447,E2 6411.447} C_VEL
LIN {X 0,Y 490.08,Z 630.238,A -85,B 0,C 180,E1 6413.262,E2 6413.262} C_VEL
LIN {X 0,Y 491.1,Z 596.023,A -85,B 0,C 180,E1 6414.386,E2 6414.386} C_VEL
LIN {X 0,Y 490.827,Z 554.52,A -85,B 0,C 180,E1 6415.089,E2 6415.089} C_VEL
LIN {X 0,Y 483.02,Z 526.81,A -85,B 0,C 180,E1 6415.932,E2 6415.932} C_VEL
LIN {X 0,Y 482.675,Z 526.81,A -85,B 0,C 180,E1 6422.231,E2 6422.231} C_VEL
LIN {X 0,Y 482.655,Z 526.81,A -85,B 0,C 180,E1 6428.863,E2 6428.863} C_VEL
LIN {X 0,Y 482.687,Z 526.81,A -85,B 0,C 180,E1 6433.837,E2 6433.837} C_VEL
LIN {X 0,Y 482.621,Z 526.81,A -85,B 0,C 180,E1 6438.851,E2 6438.851} C_VEL
LIN {X 0,Y 482.686,Z 526.81,A -85,B 0,C 180,E1 6445.633,E2 6445.633} C_VEL
LIN {X 0,Y 482.715,Z 526.81,A -85,B 0,C 180,E1 6451.942,E2 6451.942} C_VEL
LIN {X 0,Y 482.879,Z 526.81,A -85,B 0,C 180,E1 6457.905,E2 6457.905} C_VEL
LIN {X 0,Y 483.058,Z 526.81,A -85,B 0,C 180,E1 6464.311,E2 6464.311} C_VEL
LIN {X 0,Y 487.738,Z 551.692,A -85,B 0,C 180,E1 6465.542,E2 6465.542} C_VEL
LIN {X 0,Y 486.844,Z 577.667,A -85,B 0,C 180,E1 6467.318,E2 6467.318} C_VEL
LIN {X 0,Y 485.846,Z 599.444,A -85,B 0,C 180,E1 6469.684,E2 6469.684} C_VEL
LIN {X 0,Y 485.136,Z 615.387,A -85,B 0,C 180,E1 6472.384,E2 6472.384} C_VEL
LIN {X 0,Y 484.725,Z 625.232,A -85,B 0,C 180,E1 6475.078,E2 6475.078} C_VEL
LIN {X 0,Y 484.411,Z 630.789,A -85,B 0,C 180,E1 6478.214,E2 6478.214} C_VEL
LIN {X 0,Y 484.381,Z 631.457,A -85,B 0,C 180,E1 6480.006,E2 6480.006} C_VEL
LIN {X 0,Y 484.408,Z 629.063,A -85,B 0,C 180,E1 6482.693,E2 6482.693} C_VEL
LIN {X 0,Y 484.658,Z 620.899,A -85,B 0,C 180,E1 6485.833,E2 6485.833} C_VEL
LIN {X 0,Y 485.084,Z 607.114,A -85,B 0,C 180,E1 6488.757,E2 6488.757} C_VEL
LIN {X 0,Y 485.895,Z 588.5,A -85,B 0,C 180,E1 6491.266,E2 6491.266} C_VEL
LIN {X 0,Y 486.787,Z 565.798,A -85,B 0,C 180,E1 6493.266,E2 6493.266} C_VEL
LIN {X 0,Y 486.552,Z 543.853,A -85,B 0,C 180,E1 6494.547,E2 6494.547} C_VEL
LIN {X 0,Y 483.027,Z 526.81,A -85,B 0,C 180,E1 6495.342,E2 6495.342} C_VEL
LIN {X 0,Y 483.007,Z 526.81,A -85,B 0,C 180,E1 6500.175,E2 6500.175} C_VEL
LIN {X 0,Y 482.844,Z 526.81,A -85,B 0,C 180,E1 6506.045,E2 6506.045} C_VEL
LIN {X 0,Y 482.7,Z 526.81,A -85,B 0,C 180,E1 6512.229,E2 6512.229} C_VEL
LIN {X 0,Y 482.6,Z 526.81,A -85,B 0,C 180,E1 6518.868,E2 6518.868} C_VEL
LIN {X 0,Y 482.598,Z 526.81,A -85,B 0,C 180,E1 6523.808,E2 6523.808} C_VEL
LIN {X 0,Y 482.669,Z 526.81,A -85,B 0,C 180,E1 6528.843,E2 6528.843} C_VEL
LIN {X 0,Y 482.638,Z 526.81,A -85,B 0,C 180,E1 6534.656,E2 6534.656} C_VEL
LIN {X 0,Y 482.745,Z 526.81,A -85,B 0,C 180,E1 6539.875,E2 6539.875} C_VEL
LIN {X 0,Y 482.892,Z 526.81,A -85,B 0,C 180,E1 6545.941,E2 6545.941} C_VEL
LIN {X 0,Y 483.061,Z 526.81,A -85,B 0,C 180,E1 6551.729,E2 6551.729} C_VEL
LIN {X 0,Y 482.977,Z 526.81,A -85,B 0,C 180,E1 6557.319,E2 6557.319} C_VEL
LIN {X 0,Y 483.326,Z 526.81,A -85,B 0,C 180,E1 6562.797,E2 6562.797} C_VEL
LIN {X 0,Y 483.58,Z 526.81,A -85,B 0,C 180,E1 6568.202,E2 6568.202} C_VEL
LIN {X 0,Y 483.515,Z 526.81,A -85,B 0,C 180,E1 6573.586,E2 6573.586} C_VEL
LIN {X 0,Y 483.25,Z 526.81,A -85,B 0,C 180,E1 6579.008,E2 6579.008} C_VEL
LIN {X 0,Y 483.124,Z 526.81,A -85,B 0,C 180,E1 6584.515,E2 6584.515} C_VEL
LIN {X 0,Y 483,Z 526.81,A -85,B 0,C 180,E1 6590.166,E2 6590.166} C_VEL
LIN {X 0,Y 482.827,Z 526.81,A -85,B 0,C 180,E1 6596.036,E2 6596.036} C_VEL
LIN {X 0,Y 482.721,Z 526.81,A -85,B 0,C 180,E1 6602.218,E2 6602.218} C_VEL
LIN {X 0,Y 482.582,Z 526.81,A -85,B 0,C 180,E1 6608.859,E2 6608.859} C_VEL
LIN {X 0,Y 482.565,Z 526.81,A -85,B 0,C 180,E1 6613.805,E2 6613.805} C_VEL
LIN {X 0,Y 482.667,Z 526.81,A -85,B 0,C 180,E1 6618.831,E2 6618.831} C_VEL
LIN {X 0,Y 482.618,Z 526.81,A -85,B 0,C 180,E1 6624.646,E2 6624.646} C_VEL
LIN {X 0,Y 482.726,Z 526.81,A -85,B 0,C 180,E1 6629.874,E2 6629.874} C_VEL
LIN {X 0,Y 482.878,Z 526.81,A -85,B 0,C 180,E1 6635.94,E2 6635.94} C_VEL
LIN {X 0,Y 483.09,Z 526.81,A -85,B 0,C 180,E1 6641.73,E2 6641.73} C_VEL
LIN {X 0,Y 482.98,Z 526.81,A -85,B 0,C 180,E1 6647.319,E2 6647.319} C_VEL
LIN {X 0,Y 483.31,Z 526.81,A -85,B 0,C 180,E1 6652.796,E2 6652.796} C_VEL
LIN {X 0,Y 483.556,Z 526.81,A -85,B 0,C 180,E1 6658.2,E2 6658.2} C_VEL
LIN {X 0,Y 483.482,Z 526.81,A -85,B 0,C 180,E1 6663.585,E2 6663.585} C_VEL
LIN {X 0,Y 483.219,Z 526.81,A -85,B 0,C 180,E1 6669.007,E2 6669.007} C_VEL
LIN {X 0,Y 483.074,Z 526.81,A -85,B 0,C 180,E1 6674.515,E2 6674.515} C_VEL
LIN {X 0,Y 482.961,Z 526.81,A -85,B 0,C 180,E1 6680.165,E2 6680.165} C_VEL
LIN {X 0,Y 482.825,Z 526.81,A -85,B 0,C 180,E1 6686.034,E2 6686.034} C_VEL
LIN {X 0,Y 482.76,Z 526.81,A -85,B 0,C 180,E1 6692.211,E2 6692.211} C_VEL
LIN {X 0,Y 482.668,Z 526.81,A -85,B 0,C 180,E1 6698.358,E2 6698.358} C_VEL
LIN {X 0,Y 482.483,Z 526.81,A -85,B 0,C 180,E1 6703.807,E2 6703.807} C_VEL
LIN {X 0,Y 482.494,Z 526.81,A -85,B 0,C 180,E1 6708.85,E2 6708.85} C_VEL
LIN {X 0,Y 482.503,Z 526.81,A -85,B 0,C 180,E1 6712.168,E2 6712.168} C_VEL
LIN {X 0,Y 478.559,Z 526.81,A -85,B 0,C 180,E1 6714.198,E2 6714.198} C_VEL
LIN {X 0,Y 474.625,Z 526.81,A -85,B 0,C 180,E1 6716.261,E2 6716.261} C_VEL
LIN {X 0,Y 474.816,Z 526.81,A -85,B 0,C 180,E1 6721.43,E2 6721.43} C_VEL
LIN {X 0,Y 475.079,Z 526.81,A -85,B 0,C 180,E1 6723.548,E2 6723.548} C_VEL
LIN {X 0,Y 484.62,Z 561.097,A -85,B 0,C 180,E1 6724.526,E2 6724.526} C_VEL
LIN {X 0,Y 484.009,Z 606.125,A -85,B 0,C 180,E1 6725.38,E2 6725.38} C_VEL
LIN {X 0,Y 482.544,Z 638.955,A -85,B 0,C 180,E1 6726.668,E2 6726.668} C_VEL
LIN {X 0,Y 480.745,Z 670.802,A -85,B 0,C 180,E1 6728.674,E2 6728.674} C_VEL
LIN {X 0,Y 478.89,Z 699.953,A -85,B 0,C 180,E1 6731.359,E2 6731.359} C_VEL
LIN {X 0,Y 477.429,Z 724.97,A -85,B 0,C 180,E1 6734.602,E2 6734.602} C_VEL
LIN {X 0,Y 476.617,Z 745.174,A -85,B 0,C 180,E1 6738.32,E2 6738.32} C_VEL
LIN {X 0,Y 476.233,Z 759.359,A -85,B 0,C 180,E1 6742.239,E2 6742.239} C_VEL
LIN {X 0,Y 476.121,Z 766.388,A -85,B 0,C 180,E1 6745.444,E2 6745.444} C_VEL
LIN {X 0,Y 476.086,Z 769.361,A -85,B 0,C 180,E1 6748.182,E2 6748.182} C_VEL
LIN {X 0,Y 476.059,Z 769.264,A -85,B 0,C 180,E1 6751.827,E2 6751.827} C_VEL
LIN {X 0,Y 476.197,Z 764.473,A -85,B 0,C 180,E1 6755.478,E2 6755.478} C_VEL
LIN {X 0,Y 476.301,Z 754.539,A -85,B 0,C 180,E1 6759.15,E2 6759.15} C_VEL
LIN {X 0,Y 476.777,Z 738.713,A -85,B 0,C 180,E1 6762.848,E2 6762.848} C_VEL
LIN {X 0,Y 477.828,Z 717.062,A -85,B 0,C 180,E1 6766.337,E2 6766.337} C_VEL
LIN {X 0,Y 479.219,Z 690.575,A -85,B 0,C 180,E1 6769.379,E2 6769.379} C_VEL
LIN {X 0,Y 480.86,Z 661.317,A -85,B 0,C 180,E1 6771.777,E2 6771.777} C_VEL
LIN {X 0,Y 482.551,Z 628.651,A -85,B 0,C 180,E1 6773.586,E2 6773.586} C_VEL
LIN {X 0,Y 483.645,Z 593.734,A -85,B 0,C 180,E1 6774.727,E2 6774.727} C_VEL
LIN {X 0,Y 483.188,Z 555.534,A -85,B 0,C 180,E1 6775.394,E2 6775.394} C_VEL
LIN {X 0,Y 475.047,Z 526.81,A -85,B 0,C 180,E1 6776.291,E2 6776.291} C_VEL
LIN {X 0,Y 474.685,Z 526.81,A -85,B 0,C 180,E1 6782.841,E2 6782.841} C_VEL
LIN {X 0,Y 474.678,Z 526.81,A -85,B 0,C 180,E1 6789.644,E2 6789.644} C_VEL
LIN {X 0,Y 474.686,Z 526.81,A -85,B 0,C 180,E1 6795.446,E2 6795.446} C_VEL
LIN {X 0,Y 474.623,Z 526.81,A -85,B 0,C 180,E1 6800.366,E2 6800.366} C_VEL
LIN {X 0,Y 474.755,Z 526.81,A -85,B 0,C 180,E1 6806.022,E2 6806.022} C_VEL
LIN {X 0,Y 474.815,Z 526.81,A -85,B 0,C 180,E1 6811.433,E2 6811.433} C_VEL
LIN {X 0,Y 474.943,Z 526.81,A -85,B 0,C 180,E1 6817.603,E2 6817.603} C_VEL
LIN {X 0,Y 475.144,Z 527.464,A -85,B 0,C 180,E1 6823.999,E2 6823.999} C_VEL
LIN {X 0,Y 480.249,Z 551.724,A -85,B 0,C 180,E1 6825.229,E2 6825.229} C_VEL
LIN {X 0,Y 479.354,Z 576.349,A -85,B 0,C 180,E1 6826.885,E2 6826.885} C_VEL
LIN {X 0,Y 478.369,Z 597.277,A -85,B 0,C 180,E1 6829.059,E2 6829.059} C_VEL
LIN {X 0,Y 477.486,Z 614.458,A -85,B 0,C 180,E1 6831.802,E2 6831.802} C_VEL
LIN {X 0,Y 477.049,Z 625.153,A -85,B 0,C 180,E1 6834.542,E2 6834.542} C_VEL
LIN {X 0,Y 476.711,Z 631.006,A -85,B 0,C 180,E1 6837.275,E2 6837.275} C_VEL
LIN {X 0,Y 476.567,Z 632.619,A -85,B 0,C 180,E1 6840.006,E2 6840.006} C_VEL
LIN {X 0,Y 476.613,Z 630.155,A -85,B 0,C 180,E1 6842.737,E2 6842.737} C_VEL
LIN {X 0,Y 476.857,Z 621.88,A -85,B 0,C 180,E1 6845.928,E2 6845.928} C_VEL
LIN {X 0,Y 477.335,Z 607.966,A -85,B 0,C 180,E1 6848.901,E2 6848.901} C_VEL
LIN {X 0,Y 478.194,Z 589.512,A -85,B 0,C 180,E1 6851.419,E2 6851.419} C_VEL
LIN {X 0,Y 479.075,Z 566.843,A -85,B 0,C 180,E1 6853.451,E2 6853.451} C_VEL
LIN {X 0,Y 478.886,Z 545.058,A -85,B 0,C 180,E1 6854.753,E2 6854.753} C_VEL
LIN {X 0,Y 475.115,Z 526.81,A -85,B 0,C 180,E1 6855.648,E2 6855.648} C_VEL
LIN {X 0,Y 475.058,Z 526.81,A -85,B 0,C 180,E1 6860.528,E2 6860.528} C_VEL
LIN {X 0,Y 474.842,Z 526.81,A -85,B 0,C 180,E1 6866.763,E2 6866.763} C_VEL
LIN {X 0,Y 474.714,Z 526.81,A -85,B 0,C 180,E1 6872.839,E2 6872.839} C_VEL
LIN {X 0,Y 474.68,Z 526.81,A -85,B 0,C 180,E1 6877.308,E2 6877.308} C_VEL
LIN {X 0,Y 474.593,Z 526.81,A -85,B 0,C 180,E1 6882.791,E2 6882.791} C_VEL
LIN {X 0,Y 474.667,Z 526.81,A -85,B 0,C 180,E1 6887.939,E2 6887.939} C_VEL
LIN {X 0,Y 474.728,Z 526.81,A -85,B 0,C 180,E1 6892.882,E2 6892.882} C_VEL
LIN {X 0,Y 474.807,Z 526.81,A -85,B 0,C 180,E1 6899.433,E2 6899.433} C_VEL
LIN {X 0,Y 474.99,Z 526.81,A -85,B 0,C 180,E1 6905.515,E2 6905.515} C_VEL
LIN {X 0,Y 475.133,Z 526.81,A -85,B 0,C 180,E1 6911.413,E2 6911.413} C_VEL
LIN {X 0,Y 475.061,Z 526.81,A -85,B 0,C 180,E1 6917.105,E2 6917.105} C_VEL
LIN {X 0,Y 475.4,Z 526.81,A -85,B 0,C 180,E1 6922.677,E2 6922.677} C_VEL
LIN {X 0,Y 475.67,Z 526.81,A -85,B 0,C 180,E1 6928.172,E2 6928.172} C_VEL
LIN {X 0,Y 475.6,Z 526.81,A -85,B 0,C 180,E1 6933.646,E2 6933.646} C_VEL
LIN {X 0,Y 475.351,Z 526.81,A -85,B 0,C 180,E1 6939.159,E2 6939.159} C_VEL
LIN {X 0,Y 475.188,Z 526.81,A -85,B 0,C 180,E1 6944.763,E2 6944.763} C_VEL
LIN {X 0,Y 475.051,Z 526.81,A -85,B 0,C 180,E1 6950.519,E2 6950.519} C_VEL
LIN {X 0,Y 474.821,Z 526.81,A -85,B 0,C 180,E1 6956.761,E2 6956.761} C_VEL
LIN {X 0,Y 474.725,Z 526.81,A -85,B 0,C 180,E1 6962.828,E2 6962.828} C_VEL
LIN {X 0,Y 474.664,Z 526.81,A -85,B 0,C 180,E1 6967.299,E2 6967.299} C_VEL
LIN {X 0,Y 474.567,Z 526.81,A -85,B 0,C 180,E1 6972.789,E2 6972.789} C_VEL
LIN {X 0,Y 474.664,Z 526.81,A -85,B 0,C 180,E1 6977.94,E2 6977.94} C_VEL
LIN {X 0,Y 474.705,Z 526.81,A -85,B 0,C 180,E1 6982.873,E2 6982.873} C_VEL
LIN {X 0,Y 474.778,Z 526.81,A -85,B 0,C 180,E1 6989.424,E2 6989.424} C_VEL
LIN {X 0,Y 474.972,Z 526.81,A -85,B 0,C 180,E1 6995.514,E2 6995.514} C_VEL
LIN {X 0,Y 475.164,Z 526.81,A -85,B 0,C 180,E1 7001.414,E2 7001.414} C_VEL
LIN {X 0,Y 475.067,Z 526.81,A -85,B 0,C 180,E1 7007.104,E2 7007.104} C_VEL
LIN {X 0,Y 475.385,Z 526.81,A -85,B 0,C 180,E1 7012.675,E2 7012.675} C_VEL
LIN {X 0,Y 475.645,Z 526.81,A -85,B 0,C 180,E1 7018.17,E2 7018.17} C_VEL
LIN {X 0,Y 475.567,Z 526.81,A -85,B 0,C 180,E1 7023.645,E2 7023.645} C_VEL
LIN {X 0,Y 475.297,Z 526.81,A -85,B 0,C 180,E1 7029.159,E2 7029.159} C_VEL
LIN {X 0,Y 475.14,Z 526.81,A -85,B 0,C 180,E1 7034.763,E2 7034.763} C_VEL
LIN {X 0,Y 475.011,Z 526.81,A -85,B 0,C 180,E1 7040.518,E2 7040.518} C_VEL
LIN {X 0,Y 474.829,Z 526.81,A -85,B 0,C 180,E1 7046.779,E2 7046.779} C_VEL
LIN {X 0,Y 474.777,Z 526.81,A -85,B 0,C 180,E1 7052.82,E2 7052.82} C_VEL
LIN {X 0,Y 474.749,Z 526.81,A -85,B 0,C 180,E1 7057.288,E2 7057.288} C_VEL
LIN {X 0,Y 474.522,Z 526.81,A -85,B 0,C 180,E1 7062.795,E2 7062.795} C_VEL
LIN {X 0,Y 474.481,Z 526.81,A -85,B 0,C 180,E1 7067.93,E2 7067.93} C_VEL
LIN {X 0,Y 474.636,Z 526.81,A -85,B 0,C 180,E1 7074.962,E2 7074.962} C_VEL
LIN {X 0,Y 474.625,Z 526.81,A -85,B 0,C 180,E1 7076.261,E2 7076.261} C_VEL
LIN {X 0,Y 473.349,Z 526.81,A -85,B 0,C 180,E1 7077.308,E2 7077.308} C_VEL
LIN {X 0,Y 466.847,Z 526.81,A -85,B 0,C 180,E1 7080.162,E2 7080.162} C_VEL
LIN {X 0,Y 466.789,Z 526.81,A -85,B 0,C 180,E1 7080.432,E2 7080.432} C_VEL
LIN {X 0,Y 467.114,Z 527.161,A -85,B 0,C 180,E1 7083.192,E2 7083.192} C_VEL
LIN {X 0,Y 477.176,Z 562.839,A -85,B 0,C 180,E1 7084.231,E2 7084.231} C_VEL
LIN {X 0,Y 476.48,Z 607.299,A -85,B 0,C 180,E1 7085.112,E2 7085.112} C_VEL
LIN {X 0,Y 474.853,Z 641.097,A -85,B 0,C 180,E1 7086.516,E2 7086.516} C_VEL
LIN {X 0,Y 472.919,Z 672.741,A -85,B 0,C 180,E1 7088.613,E2 7088.613} C_VEL
LIN {X 0,Y 471.017,Z 701.369,A -85,B 0,C 180,E1 7091.362,E2 7091.362} C_VEL
LIN {X 0,Y 469.547,Z 725.195,A -85,B 0,C 180,E1 7094.577,E2 7094.577} C_VEL
LIN {X 0,Y 468.745,Z 745.01,A -85,B 0,C 180,E1 7098.358,E2 7098.358} C_VEL
LIN {X 0,Y 468.383,Z 758.241,A -85,B 0,C 180,E1 7102.108,E2 7102.108} C_VEL
LIN {X 0,Y 468.284,Z 765.29,A -85,B 0,C 180,E1 7105.368,E2 7105.368} C_VEL
LIN {X 0,Y 468.261,Z 768.272,A -85,B 0,C 180,E1 7108.151,E2 7108.151} C_VEL
LIN {X 0,Y 468.241,Z 768.151,A -85,B 0,C 180,E1 7111.857,E2 7111.857} C_VEL
LIN {X 0,Y 468.371,Z 763.301,A -85,B 0,C 180,E1 7115.57,E2 7115.57} C_VEL
LIN {X 0,Y 468.454,Z 753.262,A -85,B 0,C 180,E1 7119.304,E2 7119.304} C_VEL
LIN {X 0,Y 468.92,Z 737.309,A -85,B 0,C 180,E1 7123.067,E2 7123.067} C_VEL
LIN {X 0,Y 470.026,Z 715.445,A -85,B 0,C 180,E1 7126.616,E2 7126.616} C_VEL
LIN {X 0,Y 471.515,Z 688.711,A -85,B 0,C 180,E1 7129.709,E2 7129.709} C_VEL
LIN {X 0,Y 473.366,Z 657.999,A -85,B 0,C 180,E1 7132.215,E2 7132.215} C_VEL
LIN {X 0,Y 475.127,Z 625.938,A -85,B 0,C 180,E1 7133.977,E2 7133.977} C_VEL
LIN {X 0,Y 476.266,Z 590.88,A -85,B 0,C 180,E1 7135.101,E2 7135.101} C_VEL
LIN {X 0,Y 475.783,Z 557.103,A -85,B 0,C 180,E1 7135.7,E2 7135.7} C_VEL
LIN {X 0,Y 467.069,Z 526.81,A -85,B 0,C 180,E1 7136.735,E2 7136.735} C_VEL
LIN {X 0,Y 466.75,Z 526.81,A -85,B 0,C 180,E1 7143.472,E2 7143.472} C_VEL
LIN {X 0,Y 466.742,Z 526.81,A -85,B 0,C 180,E1 7150.455,E2 7150.455} C_VEL
LIN {X 0,Y 466.771,Z 526.81,A -85,B 0,C 180,E1 7157.075,E2 7157.075} C_VEL
LIN {X 0,Y 466.759,Z 526.81,A -85,B 0,C 180,E1 7164.196,E2 7164.196} C_VEL
LIN {X 0,Y 466.855,Z 526.81,A -85,B 0,C 180,E1 7168.75,E2 7168.75} C_VEL
LIN {X 0,Y 466.97,Z 526.81,A -85,B 0,C 180,E1 7175.22,E2 7175.22} C_VEL
LIN {X 0,Y 467.083,Z 526.81,A -85,B 0,C 180,E1 7181.093,E2 7181.093} C_VEL
LIN {X 0,Y 467.18,Z 527.021,A -85,B 0,C 180,E1 7183.6,E2 7183.6} C_VEL
LIN {X 0,Y 472.802,Z 552.596,A -85,B 0,C 180,E1 7184.936,E2 7184.936} C_VEL
LIN {X 0,Y 471.81,Z 577.789,A -85,B 0,C 180,E1 7186.671,E2 7186.671} C_VEL
LIN {X 0,Y 470.682,Z 599.631,A -85,B 0,C 180,E1 7189.019,E2 7189.019} C_VEL
LIN {X 0,Y 469.778,Z 615.762,A -85,B 0,C 180,E1 7191.667,E2 7191.667} C_VEL
LIN {X 0,Y 469.304,Z 626.407,A -85,B 0,C 180,E1 7194.452,E2 7194.452} C_VEL
LIN {X 0,Y 468.926,Z 632.214,A -85,B 0,C 180,E1 7197.23,E2 7197.23} C_VEL
LIN {X 0,Y 468.783,Z 633.777,A -85,B 0,C 180,E1 7200.006,E2 7200.006} C_VEL
LIN {X 0,Y 468.81,Z 631.248,A -85,B 0,C 180,E1 7202.782,E2 7202.782} C_VEL
LIN {X 0,Y 469.078,Z 622.866,A -85,B 0,C 180,E1 7206.027,E2 7206.027} C_VEL
LIN {X 0,Y 469.591,Z 608.831,A -85,B 0,C 180,E1 7209.049,E2 7209.049} C_VEL
LIN {X 0,Y 470.494,Z 590.242,A -85,B 0,C 180,E1 7211.608,E2 7211.608} C_VEL
LIN {X 0,Y 471.451,Z 567.017,A -85,B 0,C 180,E1 7213.706,E2 7213.706} C_VEL
LIN {X 0,Y 471.265,Z 546.471,A -85,B 0,C 180,E1 7214.954,E2 7214.954} C_VEL
LIN {X 0,Y 467.203,Z 526.81,A -85,B 0,C 180,E1 7215.873,E2 7215.873} C_VEL
LIN {X 0,Y 467.129,Z 526.81,A -85,B 0,C 180,E1 7220.893,E2 7220.893} C_VEL
LIN {X 0,Y 466.909,Z 526.81,A -85,B 0,C 180,E1 7227.005,E2 7227.005} C_VEL
LIN {X 0,Y 466.783,Z 526.81,A -85,B 0,C 180,E1 7233.469,E2 7233.469} C_VEL
LIN {X 0,Y 466.655,Z 526.81,A -85,B 0,C 180,E1 7240.464,E2 7240.464} C_VEL
LIN {X 0,Y 466.779,Z 526.81,A -85,B 0,C 180,E1 7247.059,E2 7247.059} C_VEL
LIN {X 0,Y 466.741,Z 526.81,A -85,B 0,C 180,E1 7251.945,E2 7251.945} C_VEL
LIN {X 0,Y 466.802,Z 526.81,A -85,B 0,C 180,E1 7258.733,E2 7258.733} C_VEL
LIN {X 0,Y 467.044,Z 526.81,A -85,B 0,C 180,E1 7265.197,E2 7265.197} C_VEL
LIN {X 0,Y 467.187,Z 526.81,A -85,B 0,C 180,E1 7271.085,E2 7271.085} C_VEL
LIN {X 0,Y 467.129,Z 526.81,A -85,B 0,C 180,E1 7276.882,E2 7276.882} C_VEL
LIN {X 0,Y 467.476,Z 526.81,A -85,B 0,C 180,E1 7282.552,E2 7282.552} C_VEL
LIN {X 0,Y 467.772,Z 526.81,A -85,B 0,C 180,E1 7288.141,E2 7288.141} C_VEL
LIN {X 0,Y 467.716,Z 526.81,A -85,B 0,C 180,E1 7293.708,E2 7293.708} C_VEL
LIN {X 0,Y 467.423,Z 526.81,A -85,B 0,C 180,E1 7299.316,E2 7299.316} C_VEL
LIN {X 0,Y 467.251,Z 526.81,A -85,B 0,C 180,E1 7305.02,E2 7305.02} C_VEL
LIN {X 0,Y 467.121,Z 526.81,A -85,B 0,C 180,E1 7310.883,E2 7310.883} C_VEL
LIN {X 0,Y 466.888,Z 526.81,A -85,B 0,C 180,E1 7316.996,E2 7316.996} C_VEL
LIN {X 0,Y 466.786,Z 526.81,A -85,B 0,C 180,E1 7323.459,E2 7323.459} C_VEL
LIN {X 0,Y 466.64,Z 526.81,A -85,B 0,C 180,E1 7330.455,E2 7330.455} C_VEL
LIN {X 0,Y 466.77,Z 526.81,A -85,B 0,C 180,E1 7337.059,E2 7337.059} C_VEL
LIN {X 0,Y 466.715,Z 526.81,A -85,B 0,C 180,E1 7341.943,E2 7341.943} C_VEL
LIN {X 0,Y 466.813,Z 526.81,A -85,B 0,C 180,E1 7348.734,E2 7348.734} C_VEL
LIN {X 0,Y 467.042,Z 526.81,A -85,B 0,C 180,E1 7355.18,E2 7355.18} C_VEL
LIN {X 0,Y 467.219,Z 526.81,A -85,B 0,C 180,E1 7361.086,E2 7361.086} C_VEL
LIN {X 0,Y 467.135,Z 526.81,A -85,B 0,C 180,E1 7366.881,E2 7366.881} C_VEL
LIN {X 0,Y 467.463,Z 526.81,A -85,B 0,C 180,E1 7372.551,E2 7372.551} C_VEL
LIN {X 0,Y 467.743,Z 526.81,A -85,B 0,C 180,E1 7378.139,E2 7378.139} C_VEL
LIN {X 0,Y 467.68,Z 526.81,A -85,B 0,C 180,E1 7383.706,E2 7383.706} C_VEL
LIN {X 0,Y 467.369,Z 526.81,A -85,B 0,C 180,E1 7389.315,E2 7389.315} C_VEL
LIN {X 0,Y 467.204,Z 526.81,A -85,B 0,C 180,E1 7395.019,E2 7395.019} C_VEL
LIN {X 0,Y 467.076,Z 526.81,A -85,B 0,C 180,E1 7400.883,E2 7400.883} C_VEL
LIN {X 0,Y 466.922,Z 526.81,A -85,B 0,C 180,E1 7406.991,E2 7406.991} C_VEL
LIN {X 0,Y 466.849,Z 526.81,A -85,B 0,C 180,E1 7413.45,E2 7413.45} C_VEL
LIN {X 0,Y 466.694,Z 526.81,A -85,B 0,C 180,E1 7418.873,E2 7418.873} C_VEL
LIN {X 0,Y 466.572,Z 526.81,A -85,B 0,C 180,E1 7425.543,E2 7425.543} C_VEL
LIN {X 0,Y 466.59,Z 526.81,A -85,B 0,C 180,E1 7431.942,E2 7431.942} C_VEL
LIN {X 0,Y 466.767,Z 526.81,A -85,B 0,C 180,E1 7438.74,E2 7438.74} C_VEL
LIN {X 0,Y 466.789,Z 526.81,A -85,B 0,C 180,E1 7440.432,E2 7440.432} C_VEL
LIN {X 0,Y 462.906,Z 526.81,A -85,B 0,C 180,E1 7441.448,E2 7441.448} C_VEL
LIN {X 0,Y 459.071,Z 526.81,A -85,B 0,C 180,E1 7442.482,E2 7442.482} C_VEL
LIN {X 0,Y 459.119,Z 526.81,A -85,B 0,C 180,E1 7442.804,E2 7442.804} C_VEL
LIN {X 0,Y 469.734,Z 564.067,A -85,B 0,C 180,E1 7443.926,E2 7443.926} C_VEL
LIN {X 0,Y 469.014,Z 606.91,A -85,B 0,C 180,E1 7444.801,E2 7444.801} C_VEL
LIN {X 0,Y 467.266,Z 640.87,A -85,B 0,C 180,E1 7446.238,E2 7446.238} C_VEL
LIN {X 0,Y 465.218,Z 672.858,A -85,B 0,C 180,E1 7448.407,E2 7448.407} C_VEL
LIN {X 0,Y 463.242,Z 700.356,A -85,B 0,C 180,E1 7451.097,E2 7451.097} C_VEL
LIN {X 0,Y 461.657,Z 725.394,A -85,B 0,C 180,E1 7454.55,E2 7454.55} C_VEL
LIN {X 0,Y 460.846,Z 744.842,A -85,B 0,C 180,E1 7458.396,E2 7458.396} C_VEL
LIN {X 0,Y 460.502,Z 758.326,A -85,B 0,C 180,E1 7462.447,E2 7462.447} C_VEL
LIN {X 0,Y 460.446,Z 765.473,A -85,B 0,C 180,E1 7466.234,E2 7466.234} C_VEL
LIN {X 0,Y 460.471,Z 767.759,A -85,B 0,C 180,E1 7470.004,E2 7470.004} C_VEL
LIN {X 0,Y 460.443,Z 765.199,A -85,B 0,C 180,E1 7473.775,E2 7473.775} C_VEL
LIN {X 0,Y 460.539,Z 757.717,A -85,B 0,C 180,E1 7477.561,E2 7477.561} C_VEL
LIN {X 0,Y 460.879,Z 743.756,A -85,B 0,C 180,E1 7481.613,E2 7481.613} C_VEL
LIN {X 0,Y 461.69,Z 723.658,A -85,B 0,C 180,E1 7485.458,E2 7485.458} C_VEL
LIN {X 0,Y 463.046,Z 699.438,A -85,B 0,C 180,E1 7488.723,E2 7488.723} C_VEL
LIN {X 0,Y 464.809,Z 671.631,A -85,B 0,C 180,E1 7491.421,E2 7491.421} C_VEL
LIN {X 0,Y 466.793,Z 639.217,A -85,B 0,C 180,E1 7493.606,E2 7493.606} C_VEL
LIN {X 0,Y 468.378,Z 606.203,A -85,B 0,C 180,E1 7495.018,E2 7495.018} C_VEL
LIN {X 0,Y 469.139,Z 564.619,A -85,B 0,C 180,E1 7495.889,E2 7495.889} C_VEL
LIN {X 0,Y 464.378,Z 543.573,A -85,B 0,C 180,E1 7496.482,E2 7496.482} C_VEL
LIN {X 0,Y 459.106,Z 526.81,A -85,B 0,C 180,E1 7497.092,E2 7497.092} C_VEL
LIN {X 0,Y 458.767,Z 526.81,A -85,B 0,C 180,E1 7504.134,E2 7504.134} C_VEL
LIN {X 0,Y 458.861,Z 526.81,A -85,B 0,C 180,E1 7510.644,E2 7510.644} C_VEL
LIN {X 0,Y 458.844,Z 526.81,A -85,B 0,C 180,E1 7516.554,E2 7516.554} C_VEL
LIN {X 0,Y 458.771,Z 526.81,A -85,B 0,C 180,E1 7522.386,E2 7522.386} C_VEL
LIN {X 0,Y 458.946,Z 526.81,A -85,B 0,C 180,E1 7529.073,E2 7529.073} C_VEL
LIN {X 0,Y 458.992,Z 526.81,A -85,B 0,C 180,E1 7534.615,E2 7534.615} C_VEL
LIN {X 0,Y 459.181,Z 526.81,A -85,B 0,C 180,E1 7540.755,E2 7540.755} C_VEL
LIN {X 0,Y 459.234,Z 526.81,A -85,B 0,C 180,E1 7543.175,E2 7543.175} C_VEL
LIN {X 0,Y 465.359,Z 553.486,A -85,B 0,C 180,E1 7544.632,E2 7544.632} C_VEL
LIN {X 0,Y 464.288,Z 579.374,A -85,B 0,C 180,E1 7546.451,E2 7546.451} C_VEL
LIN {X 0,Y 463.099,Z 600.658,A -85,B 0,C 180,E1 7548.785,E2 7548.785} C_VEL
LIN {X 0,Y 462.071,Z 617.065,A -85,B 0,C 180,E1 7551.527,E2 7551.527} C_VEL
LIN {X 0,Y 461.539,Z 627.685,A -85,B 0,C 180,E1 7554.358,E2 7554.358} C_VEL
LIN {X 0,Y 461.149,Z 633.45,A -85,B 0,C 180,E1 7557.183,E2 7557.183} C_VEL
LIN {X 0,Y 460.972,Z 634.951,A -85,B 0,C 180,E1 7560.006,E2 7560.006} C_VEL
LIN {X 0,Y 461.004,Z 632.337,A -85,B 0,C 180,E1 7562.829,E2 7562.829} C_VEL
LIN {X 0,Y 461.278,Z 623.847,A -85,B 0,C 180,E1 7566.129,E2 7566.129} C_VEL
LIN {X 0,Y 461.852,Z 609.674,A -85,B 0,C 180,E1 7569.202,E2 7569.202} C_VEL
LIN {X 0,Y 462.807,Z 590.945,A -85,B 0,C 180,E1 7571.804,E2 7571.804} C_VEL
LIN {X 0,Y 463.861,Z 567.131,A -85,B 0,C 180,E1 7573.969,E2 7573.969} C_VEL
LIN {X 0,Y 463.677,Z 548.023,A -85,B 0,C 180,E1 7575.148,E2 7575.148} C_VEL
LIN {X 0,Y 459.267,Z 526.81,A -85,B 0,C 180,E1 7576.159,E2 7576.159} C_VEL
LIN {X 0,Y 459.144,Z 526.81,A -85,B 0,C 180,E1 7582.572,E2 7582.572} C_VEL
LIN {X 0,Y 458.977,Z 526.81,A -85,B 0,C 180,E1 7587.51,E2 7587.51} C_VEL
LIN {X 0,Y 458.792,Z 526.81,A -85,B 0,C 180,E1 7594.131,E2 7594.131} C_VEL
LIN {X 0,Y 458.743,Z 526.81,A -85,B 0,C 180,E1 7600.608,E2 7600.608} C_VEL
LIN {X 0,Y 458.85,Z 526.81,A -85,B 0,C 180,E1 7606.552,E2 7606.552} C_VEL
LIN {X 0,Y 458.81,Z 526.81,A -85,B 0,C 180,E1 7612.378,E2 7612.378} C_VEL
LIN {X 0,Y 458.887,Z 526.81,A -85,B 0,C 180,E1 7619.083,E2 7619.083} C_VEL
LIN {X 0,Y 459.053,Z 526.81,A -85,B 0,C 180,E1 7624.605,E2 7624.605} C_VEL
LIN {X 0,Y 459.282,Z 526.81,A -85,B 0,C 180,E1 7630.747,E2 7630.747} C_VEL
LIN {X 0,Y 459.23,Z 526.81,A -85,B 0,C 180,E1 7636.652,E2 7636.652} C_VEL
LIN {X 0,Y 459.548,Z 526.81,A -85,B 0,C 180,E1 7642.423,E2 7642.423} C_VEL
LIN {X 0,Y 459.86,Z 526.81,A -85,B 0,C 180,E1 7648.109,E2 7648.109} C_VEL
LIN {X 0,Y 459.798,Z 526.81,A -85,B 0,C 180,E1 7653.772,E2 7653.772} C_VEL
LIN {X 0,Y 459.522,Z 526.81,A -85,B 0,C 180,E1 7659.478,E2 7659.478} C_VEL
LIN {X 0,Y 459.317,Z 526.81,A -85,B 0,C 180,E1 7665.286,E2 7665.286} C_VEL
LIN {X 0,Y 459.161,Z 526.81,A -85,B 0,C 180,E1 7671.263,E2 7671.263} C_VEL
LIN {X 0,Y 458.956,Z 526.81,A -85,B 0,C 180,E1 7677.502,E2 7677.502} C_VEL
LIN {X 0,Y 458.792,Z 526.81,A -85,B 0,C 180,E1 7684.121,E2 7684.121} C_VEL
LIN {X 0,Y 458.727,Z 526.81,A -85,B 0,C 180,E1 7690.607,E2 7690.607} C_VEL
LIN {X 0,Y 458.831,Z 526.81,A -85,B 0,C 180,E1 7696.543,E2 7696.543} C_VEL
LIN {X 0,Y 458.785,Z 526.81,A -85,B 0,C 180,E1 7702.369,E2 7702.369} C_VEL
LIN {X 0,Y 458.887,Z 526.81,A -85,B 0,C 180,E1 7709.068,E2 7709.068} C_VEL
LIN {X 0,Y 459.05,Z 526.81,A -85,B 0,C 180,E1 7714.605,E2 7714.605} C_VEL
LIN {X 0,Y 459.307,Z 526.81,A -85,B 0,C 180,E1 7720.748,E2 7720.748} C_VEL
LIN {X 0,Y 459.229,Z 526.81,A -85,B 0,C 180,E1 7726.651,E2 7726.651} C_VEL
LIN {X 0,Y 459.538,Z 526.81,A -85,B 0,C 180,E1 7732.421,E2 7732.421} C_VEL
LIN {X 0,Y 459.832,Z 526.81,A -85,B 0,C 180,E1 7738.107,E2 7738.107} C_VEL
LIN {X 0,Y 459.763,Z 526.81,A -85,B 0,C 180,E1 7743.77,E2 7743.77} C_VEL
LIN {X 0,Y 459.466,Z 526.81,A -85,B 0,C 180,E1 7749.477,E2 7749.477} C_VEL
LIN {X 0,Y 459.27,Z 526.81,A -85,B 0,C 180,E1 7755.285,E2 7755.285} C_VEL
LIN {X 0,Y 459.12,Z 526.81,A -85,B 0,C 180,E1 7761.262,E2 7761.262} C_VEL
LIN {X 0,Y 458.977,Z 526.81,A -85,B 0,C 180,E1 7767.497,E2 7767.497} C_VEL
LIN {X 0,Y 458.864,Z 526.81,A -85,B 0,C 180,E1 7774.111,E2 7774.111} C_VEL
LIN {X 0,Y 458.754,Z 526.81,A -85,B 0,C 180,E1 7780.623,E2 7780.623} C_VEL
LIN {X 0,Y 458.634,Z 526.81,A -85,B 0,C 180,E1 7786.564,E2 7786.564} C_VEL
LIN {X 0,Y 458.671,Z 526.81,A -85,B 0,C 180,E1 7792.382,E2 7792.382} C_VEL
LIN {X 0,Y 458.85,Z 526.81,A -85,B 0,C 180,E1 7799.068,E2 7799.068} C_VEL
LIN {X 0,Y 459.071,Z 526.81,A -85,B 0,C 180,E1 7802.482,E2 7802.482} C_VEL
LIN {X 0,Y 461.187,Z 529.773,A -85,B 0,C 180,E1 7802.949,E2 7802.949} C_VEL
LIN {X 0,Y 463.661,Z 539.755,A -85,B 0,C 180,E1 7803.25,E2 7803.25} C_VEL
LIN {X 0,Y 461.326,Z 559.633,A -85,B 0,C 180,E1 7803.48,E2 7803.48} C_VEL
LIN {X 0,Y 461.629,Z 560.883,A -85,B 0,C 180,E1 7803.515,E2 7803.515} C_VEL
LIN {X 0,Y 461.623,Z 604.571,A -85,B 0,C 180,E1 7804.425,E2 7804.425} C_VEL
LIN {X 0,Y 459.85,Z 638.361,A -85,B 0,C 180,E1 7805.831,E2 7805.831} C_VEL
LIN {X 0,Y 457.679,Z 669.952,A -85,B 0,C 180,E1 7807.944,E2 7807.944} C_VEL
LIN {X 0,Y 455.563,Z 698.435,A -85,B 0,C 180,E1 7810.728,E2 7810.728} C_VEL
LIN {X 0,Y 453.977,Z 722.525,A -85,B 0,C 180,E1 7814.034,E2 7814.034} C_VEL
LIN {X 0,Y 453.053,Z 741.583,A -85,B 0,C 180,E1 7817.704,E2 7817.704} C_VEL
LIN {X 0,Y 452.653,Z 756.065,A -85,B 0,C 180,E1 7821.862,E2 7821.862} C_VEL
LIN {X 0,Y 452.598,Z 763.086,A -85,B 0,C 180,E1 7825.207,E2 7825.207} C_VEL
LIN {X 0,Y 452.606,Z 766.092,A -85,B 0,C 180,E1 7828.088,E2 7828.088} C_VEL
LIN {X 0,Y 452.589,Z 765.926,A -85,B 0,C 180,E1 7831.922,E2 7831.922} C_VEL
LIN {X 0,Y 452.712,Z 760.959,A -85,B 0,C 180,E1 7835.763,E2 7835.763} C_VEL
LIN {X 0,Y 452.755,Z 750.708,A -85,B 0,C 180,E1 7839.63,E2 7839.63} C_VEL
LIN {X 0,Y 453.25,Z 734.521,A -85,B 0,C 180,E1 7843.527,E2 7843.527} C_VEL
LIN {X 0,Y 454.411,Z 712.32,A -85,B 0,C 180,E1 7847.205,E2 7847.205} C_VEL
LIN {X 0,Y 456.216,Z 685.195,A -85,B 0,C 180,E1 7850.398,E2 7850.398} C_VEL
LIN {X 0,Y 458.284,Z 655.002,A -85,B 0,C 180,E1 7852.907,E2 7852.907} C_VEL
LIN {X 0,Y 460.295,Z 622.126,A -85,B 0,C 180,E1 7854.736,E2 7854.736} C_VEL
LIN {X 0,Y 461.513,Z 589.543,A -85,B 0,C 180,E1 7855.804,E2 7855.804} C_VEL
LIN {X 0,Y 461.166,Z 560.501,A -85,B 0,C 180,E1 7856.357,E2 7856.357} C_VEL
LIN {X 0,Y 451.099,Z 526.81,A -85,B 0,C 180,E1 7857.583,E2 7857.583} C_VEL
LIN {X 0,Y 450.833,Z 526.81,A -85,B 0,C 180,E1 7864.82,E2 7864.82} C_VEL
LIN {X 0,Y 450.895,Z 526.81,A -85,B 0,C 180,E1 7869.649,E2 7869.649} C_VEL
LIN {X 0,Y 450.861,Z 526.81,A -85,B 0,C 180,E1 7875.164,E2 7875.164} C_VEL
LIN {X 0,Y 450.869,Z 526.81,A -85,B 0,C 180,E1 7880.574,E2 7880.574} C_VEL
LIN {X 0,Y 450.952,Z 526.81,A -85,B 0,C 180,E1 7887.516,E2 7887.516} C_VEL
LIN {X 0,Y 451.087,Z 526.81,A -85,B 0,C 180,E1 7894.137,E2 7894.137} C_VEL
LIN {X 0,Y 451.224,Z 526.81,A -85,B 0,C 180,E1 7900.402,E2 7900.402} C_VEL
LIN {X 0,Y 451.29,Z 526.81,A -85,B 0,C 180,E1 7902.736,E2 7902.736} C_VEL
LIN {X 0,Y 457.931,Z 554.123,A -85,B 0,C 180,E1 7904.284,E2 7904.284} C_VEL
LIN {X 0,Y 456.823,Z 579.686,A -85,B 0,C 180,E1 7906.103,E2 7906.103} C_VEL
LIN {X 0,Y 455.537,Z 601.455,A -85,B 0,C 180,E1 7908.503,E2 7908.503} C_VEL
LIN {X 0,Y 454.407,Z 618.457,A -85,B 0,C 180,E1 7911.383,E2 7911.383} C_VEL
LIN {X 0,Y 453.8,Z 628.981,A -85,B 0,C 180,E1 7914.262,E2 7914.262} C_VEL
LIN {X 0,Y 453.368,Z 634.687,A -85,B 0,C 180,E1 7917.135,E2 7917.135} C_VEL
LIN {X 0,Y 453.178,Z 636.124,A -85,B 0,C 180,E1 7920.006,E2 7920.006} C_VEL
LIN {X 0,Y 453.192,Z 633.422,A -85,B 0,C 180,E1 7922.878,E2 7922.878} C_VEL
LIN {X 0,Y 453.479,Z 624.784,A -85,B 0,C 180,E1 7926.235,E2 7926.235} C_VEL
LIN {X 0,Y 454.101,Z 610.438,A -85,B 0,C 180,E1 7929.36,E2 7929.36} C_VEL
LIN {X 0,Y 455.082,Z 591.533,A -85,B 0,C 180,E1 7932.007,E2 7932.007} C_VEL
LIN {X 0,Y 456.168,Z 567.976,A -85,B 0,C 180,E1 7934.174,E2 7934.174} C_VEL
LIN {X 0,Y 456.135,Z 549.902,A -85,B 0,C 180,E1 7935.319,E2 7935.319} C_VEL
LIN {X 0,Y 451.349,Z 526.81,A -85,B 0,C 180,E1 7936.45,E2 7936.45} C_VEL
LIN {X 0,Y 451.242,Z 526.81,A -85,B 0,C 180,E1 7941.664,E2 7941.664} C_VEL
LIN {X 0,Y 450.995,Z 526.81,A -85,B 0,C 180,E1 7948.04,E2 7948.04} C_VEL
LIN {X 0,Y 450.852,Z 526.81,A -85,B 0,C 180,E1 7954.818,E2 7954.818} C_VEL
LIN {X 0,Y 450.821,Z 526.81,A -85,B 0,C 180,E1 7959.656,E2 7959.656} C_VEL
LIN {X 0,Y 450.82,Z 526.81,A -85,B 0,C 180,E1 7965.142,E2 7965.142} C_VEL
LIN {X 0,Y 450.901,Z 526.81,A -85,B 0,C 180,E1 7970.567,E2 7970.567} C_VEL
LIN {X 0,Y 450.877,Z 526.81,A -85,B 0,C 180,E1 7977.095,E2 7977.095} C_VEL
LIN {X 0,Y 451.145,Z 526.81,A -85,B 0,C 180,E1 7984.128,E2 7984.128} C_VEL
LIN {X 0,Y 451.325,Z 526.81,A -85,B 0,C 180,E1 7990.394,E2 7990.394} C_VEL
LIN {X 0,Y 451.352,Z 526.81,A -85,B 0,C 180,E1 7996.621,E2 7996.621} C_VEL
LIN {X 0,Y 451.654,Z 526.81,A -85,B 0,C 180,E1 8002.289,E2 8002.289} C_VEL
LIN {X 0,Y 451.968,Z 526.81,A -85,B 0,C 180,E1 8008.076,E2 8008.076} C_VEL
LIN {X 0,Y 451.9,Z 526.81,A -85,B 0,C 180,E1 8013.838,E2 8013.838} C_VEL
LIN {X 0,Y 451.59,Z 526.81,A -85,B 0,C 180,E1 8019.646,E2 8019.646} C_VEL
LIN {X 0,Y 451.388,Z 526.81,A -85,B 0,C 180,E1 8025.561,E2 8025.561} C_VEL
LIN {X 0,Y 451.225,Z 526.81,A -85,B 0,C 180,E1 8031.655,E2 8031.655} C_VEL
LIN {X 0,Y 450.972,Z 526.81,A -85,B 0,C 180,E1 8038.031,E2 8038.031} C_VEL
LIN {X 0,Y 450.847,Z 526.81,A -85,B 0,C 180,E1 8044.808,E2 8044.808} C_VEL
LIN {X 0,Y 450.797,Z 526.81,A -85,B 0,C 180,E1 8049.647,E2 8049.647} C_VEL
LIN {X 0,Y 450.806,Z 526.81,A -85,B 0,C 180,E1 8055.141,E2 8055.141} C_VEL
LIN {X 0,Y 450.887,Z 526.81,A -85,B 0,C 180,E1 8060.557,E2 8060.557} C_VEL
LIN {X 0,Y 450.896,Z 526.81,A -85,B 0,C 180,E1 8067.497,E2 8067.497} C_VEL
LIN {X 0,Y 451.128,Z 526.81,A -85,B 0,C 180,E1 8074.127,E2 8074.127} C_VEL
LIN {X 0,Y 451.348,Z 526.81,A -85,B 0,C 180,E1 8080.395,E2 8080.395} C_VEL
LIN {X 0,Y 451.329,Z 526.81,A -85,B 0,C 180,E1 8086.601,E2 8086.601} C_VEL
LIN {X 0,Y 451.646,Z 526.81,A -85,B 0,C 180,E1 8092.288,E2 8092.288} C_VEL
LIN {X 0,Y 451.937,Z 526.81,A -85,B 0,C 180,E1 8098.074,E2 8098.074} C_VEL
LIN {X 0,Y 451.862,Z 526.81,A -85,B 0,C 180,E1 8103.836,E2 8103.836} C_VEL
LIN {X 0,Y 451.534,Z 526.81,A -85,B 0,C 180,E1 8109.645,E2 8109.645} C_VEL
LIN {X 0,Y 451.342,Z 526.81,A -85,B 0,C 180,E1 8115.56,E2 8115.56} C_VEL
LIN {X 0,Y 451.186,Z 526.81,A -85,B 0,C 180,E1 8121.655,E2 8121.655} C_VEL
LIN {X 0,Y 451,Z 526.81,A -85,B 0,C 180,E1 8128.026,E2 8128.026} C_VEL
LIN {X 0,Y 450.942,Z 526.81,A -85,B 0,C 180,E1 8134.796,E2 8134.796} C_VEL
LIN {X 0,Y 450.84,Z 526.81,A -85,B 0,C 180,E1 8139.639,E2 8139.639} C_VEL
LIN {X 0,Y 450.657,Z 526.81,A -85,B 0,C 180,E1 8145.134,E2 8145.134} C_VEL
LIN {X 0,Y 450.742,Z 526.81,A -85,B 0,C 180,E1 8150.574,E2 8150.574} C_VEL
LIN {X 0,Y 450.814,Z 526.81,A -85,B 0,C 180,E1 8157.085,E2 8157.085} C_VEL
LIN {X 0,Y 451.159,Z 526.81,A -85,B 0,C 180,E1 8162.43,E2 8162.43} C_VEL
LIN {X 0,Y 461.629,Z 560.883,A -85,B 0,C 180,E1 8163.515,E2 8163.515} C_VEL
LIN {X 0,Y 461.448,Z 571.503,A -85,B 0,C 180,E1 8163.682,E2 8163.682} C_VEL
LIN {X 0,Y 454.653,Z 592.993,A -85,B 0,C 180,E1 8163.799,E2 8163.799} C_VEL
LIN {X 0,Y 454.492,Z 595.213,A -85,B 0,C 180,E1 8163.851,E2 8163.851} C_VEL
LIN {X 0,Y 452.785,Z 629.531,A -85,B 0,C 180,E1 8165.1,E2 8165.1} C_VEL
LIN {X 0,Y 450.627,Z 660.537,A -85,B 0,C 180,E1 8166.98,E2 8166.98} C_VEL
LIN {X 0,Y 448.418,Z 690.003,A -85,B 0,C 180,E1 8169.628,E2 8169.628} C_VEL
LIN {X 0,Y 446.573,Z 714.699,A -85,B 0,C 180,E1 8172.748,E2 8172.748} C_VEL
LIN {X 0,Y 445.317,Z 735.855,A -85,B 0,C 180,E1 8176.487,E2 8176.487} C_VEL
LIN {X 0,Y 444.832,Z 750.451,A -85,B 0,C 180,E1 8180.206,E2 8180.206} C_VEL
LIN {X 0,Y 444.777,Z 760.346,A -85,B 0,C 180,E1 8184.143,E2 8184.143} C_VEL
LIN {X 0,Y 444.781,Z 764.992,A -85,B 0,C 180,E1 8188.054,E2 8188.054} C_VEL
LIN {X 0,Y 444.765,Z 764.806,A -85,B 0,C 180,E1 8191.955,E2 8191.955} C_VEL
LIN {X 0,Y 444.881,Z 759.787,A -85,B 0,C 180,E1 8195.865,E2 8195.865} C_VEL
LIN {X 0,Y 444.889,Z 749.446,A -85,B 0,C 180,E1 8199.802,E2 8199.802} C_VEL
LIN {X 0,Y 445.446,Z 733.164,A -85,B 0,C 180,E1 8203.769,E2 8203.769} C_VEL
LIN {X 0,Y 446.646,Z 710.828,A -85,B 0,C 180,E1 8207.513,E2 8207.513} C_VEL
LIN {X 0,Y 448.497,Z 684.77,A -85,B 0,C 180,E1 8210.636,E2 8210.636} C_VEL
LIN {X 0,Y 450.667,Z 654.644,A -85,B 0,C 180,E1 8213.206,E2 8213.206} C_VEL
LIN {X 0,Y 452.819,Z 621.906,A -85,B 0,C 180,E1 8215.077,E2 8215.077} C_VEL
LIN {X 0,Y 454.193,Z 588.576,A -85,B 0,C 180,E1 8216.196,E2 8216.196} C_VEL
LIN {X 0,Y 453.858,Z 561.803,A -85,B 0,C 180,E1 8216.726,E2 8216.726} C_VEL
LIN {X 0,Y 444.475,Z 531.212,A -85,B 0,C 180,E1 8217.852,E2 8217.852} C_VEL
LIN {X 0,Y 443.115,Z 526.81,A -85,B 0,C 180,E1 8218.106,E2 8218.106} C_VEL
LIN {X 0,Y 442.929,Z 526.81,A -85,B 0,C 180,E1 8224.891,E2 8224.891} C_VEL
LIN {X 0,Y 442.89,Z 526.81,A -85,B 0,C 180,E1 8231.24,E2 8231.24} C_VEL
LIN {X 0,Y 442.864,Z 526.81,A -85,B 0,C 180,E1 8236.873,E2 8236.873} C_VEL
LIN {X 0,Y 442.894,Z 526.81,A -85,B 0,C 180,E1 8242.033,E2 8242.033} C_VEL
LIN {X 0,Y 443.006,Z 526.81,A -85,B 0,C 180,E1 8248.706,E2 8248.706} C_VEL
LIN {X 0,Y 443.163,Z 526.81,A -85,B 0,C 180,E1 8255.804,E2 8255.804} C_VEL
LIN {X 0,Y 443.338,Z 526.81,A -85,B 0,C 180,E1 8262.228,E2 8262.228} C_VEL
LIN {X 0,Y 450.451,Z 555.171,A -85,B 0,C 180,E1 8263.94,E2 8263.94} C_VEL
LIN {X 0,Y 449.352,Z 581.484,A -85,B 0,C 180,E1 8265.867,E2 8265.867} C_VEL
LIN {X 0,Y 447.96,Z 602.998,A -85,B 0,C 180,E1 8268.306,E2 8268.306} C_VEL
LIN {X 0,Y 446.722,Z 619.857,A -85,B 0,C 180,E1 8271.234,E2 8271.234} C_VEL
LIN {X 0,Y 446.069,Z 630.323,A -85,B 0,C 180,E1 8274.162,E2 8274.162} C_VEL
LIN {X 0,Y 445.611,Z 635.948,A -85,B 0,C 180,E1 8277.085,E2 8277.085} C_VEL
LIN {X 0,Y 445.367,Z 637.302,A -85,B 0,C 180,E1 8280.006,E2 8280.006} C_VEL
LIN {X 0,Y 445.405,Z 634.502,A -85,B 0,C 180,E1 8282.929,E2 8282.929} C_VEL
LIN {X 0,Y 445.678,Z 625.729,A -85,B 0,C 180,E1 8286.345,E2 8286.345} C_VEL
LIN {X 0,Y 446.356,Z 611.214,A -85,B 0,C 180,E1 8289.524,E2 8289.524} C_VEL
LIN {X 0,Y 447.384,Z 592.114,A -85,B 0,C 180,E1 8292.217,E2 8292.217} C_VEL
LIN {X 0,Y 448.521,Z 568.706,A -85,B 0,C 180,E1 8294.394,E2 8294.394} C_VEL
LIN {X 0,Y 448.286,Z 550.11,A -85,B 0,C 180,E1 8295.594,E2 8295.594} C_VEL
LIN {X 0,Y 443.419,Z 526.81,A -85,B 0,C 180,E1 8296.735,E2 8296.735} C_VEL
LIN {X 0,Y 443.224,Z 526.81,A -85,B 0,C 180,E1 8302.719,E2 8302.719} C_VEL
LIN {X 0,Y 443.053,Z 526.81,A -85,B 0,C 180,E1 8308.588,E2 8308.588} C_VEL
LIN {X 0,Y 442.925,Z 526.81,A -85,B 0,C 180,E1 8315.534,E2 8315.534} C_VEL
LIN {X 0,Y 442.79,Z 526.81,A -85,B 0,C 180,E1 8321.206,E2 8321.206} C_VEL
LIN {X 0,Y 442.867,Z 526.81,A -85,B 0,C 180,E1 8326.856,E2 8326.856} C_VEL
LIN {X 0,Y 442.926,Z 526.81,A -85,B 0,C 180,E1 8332.02,E2 8332.02} C_VEL
LIN {X 0,Y 442.968,Z 526.81,A -85,B 0,C 180,E1 8338.711,E2 8338.711} C_VEL
LIN {X 0,Y 443.159,Z 526.81,A -85,B 0,C 180,E1 8343.626,E2 8343.626} C_VEL
LIN {X 0,Y 443.397,Z 526.81,A -85,B 0,C 180,E1 8350.029,E2 8350.029} C_VEL
LIN {X 0,Y 443.366,Z 526.81,A -85,B 0,C 180,E1 8356.165,E2 8356.165} C_VEL
LIN {X 0,Y 443.722,Z 526.81,A -85,B 0,C 180,E1 8362.151,E2 8362.151} C_VEL
LIN {X 0,Y 444.055,Z 526.81,A -85,B 0,C 180,E1 8368.041,E2 8368.041} C_VEL
LIN {X 0,Y 443.981,Z 526.81,A -85,B 0,C 180,E1 8373.906,E2 8373.906} C_VEL
LIN {X 0,Y 443.675,Z 526.81,A -85,B 0,C 180,E1 8379.82,E2 8379.82} C_VEL
LIN {X 0,Y 443.45,Z 526.81,A -85,B 0,C 180,E1 8385.847,E2 8385.847} C_VEL
LIN {X 0,Y 443.258,Z 526.81,A -85,B 0,C 180,E1 8392.065,E2 8392.065} C_VEL
LIN {X 0,Y 443.028,Z 526.81,A -85,B 0,C 180,E1 8398.579,E2 8398.579} C_VEL
LIN {X 0,Y 442.913,Z 526.81,A -85,B 0,C 180,E1 8405.525,E2 8405.525} C_VEL
LIN {X 0,Y 442.772,Z 526.81,A -85,B 0,C 180,E1 8411.205,E2 8411.205} C_VEL
LIN {X 0,Y 442.858,Z 526.81,A -85,B 0,C 180,E1 8416.855,E2 8416.855} C_VEL
LIN {X 0,Y 442.903,Z 526.81,A -85,B 0,C 180,E1 8422.019,E2 8422.019} C_VEL
LIN {X 0,Y 442.959,Z 526.81,A -85,B 0,C 180,E1 8428.698,E2 8428.698} C_VEL
LIN {X 0,Y 443.223,Z 526.81,A -85,B 0,C 180,E1 8435.795,E2 8435.795} C_VEL
LIN {X 0,Y 443.431,Z 526.81,A -85,B 0,C 180,E1 8442.098,E2 8442.098} C_VEL
LIN {X 0,Y 443.452,Z 526.81,A -85,B 0,C 180,E1 8448.173,E2 8448.173} C_VEL
LIN {X 0,Y 443.8,Z 526.81,A -85,B 0,C 180,E1 8454.12,E2 8454.12} C_VEL
LIN {X 0,Y 444.015,Z 526.81,A -85,B 0,C 180,E1 8459.994,E2 8459.994} C_VEL
LIN {X 0,Y 443.724,Z 526.81,A -85,B 0,C 180,E1 8465.869,E2 8465.869} C_VEL
LIN {X 0,Y 443.494,Z 526.81,A -85,B 0,C 180,E1 8471.813,E2 8471.813} C_VEL
LIN {X 0,Y 443.375,Z 526.81,A -85,B 0,C 180,E1 8477.892,E2 8477.892} C_VEL
LIN {X 0,Y 443.183,Z 526.81,A -85,B 0,C 180,E1 8484.194,E2 8484.194} C_VEL
LIN {X 0,Y 443.008,Z 526.81,A -85,B 0,C 180,E1 8490.832,E2 8490.832} C_VEL
LIN {X 0,Y 443.023,Z 526.81,A -85,B 0,C 180,E1 8495.511,E2 8495.511} C_VEL
LIN {X 0,Y 442.766,Z 526.81,A -85,B 0,C 180,E1 8501.217,E2 8501.217} C_VEL
LIN {X 0,Y 442.672,Z 526.81,A -85,B 0,C 180,E1 8506.845,E2 8506.845} C_VEL
LIN {X 0,Y 442.786,Z 526.81,A -85,B 0,C 180,E1 8512.018,E2 8512.018} C_VEL
LIN {X 0,Y 442.923,Z 526.81,A -85,B 0,C 180,E1 8518.698,E2 8518.698} C_VEL
LIN {X 0,Y 443.182,Z 526.81,A -85,B 0,C 180,E1 8522.029,E2 8522.029} C_VEL
LIN {X 0,Y 454.878,Z 565.505,A -85,B 0,C 180,E1 8523.288,E2 8523.288} C_VEL
LIN {X 0,Y 454.492,Z 595.213,A -85,B 0,C 180,E1 8523.851,E2 8523.851} C_VEL
LIN {X 0,Y 450.091,Z 611.95,A -85,B 0,C 180,E1 8524.204,E2 8524.204} C_VEL
LIN {X 0,Y 445.296,Z 628.247,A -85,B 0,C 180,E1 8524.75,E2 8524.75} C_VEL
LIN {X 0,Y 442.921,Z 660.934,A -85,B 0,C 180,E1 8526.774,E2 8526.774} C_VEL
LIN {X 0,Y 440.594,Z 690.552,A -85,B 0,C 180,E1 8529.512,E2 8529.512} C_VEL
LIN {X 0,Y 438.599,Z 716.513,A -85,B 0,C 180,E1 8532.942,E2 8532.942} C_VEL
LIN {X 0,Y 437.404,Z 736.827,A -85,B 0,C 180,E1 8536.748,E2 8536.748} C_VEL
LIN {X 0,Y 436.959,Z 751.638,A -85,B 0,C 180,E1 8540.82,E2 8540.82} C_VEL
LIN {X 0,Y 436.94,Z 760.839,A -85,B 0,C 180,E1 8545.035,E2 8545.035} C_VEL
LIN {X 0,Y 436.955,Z 763.881,A -85,B 0,C 180,E1 8548.019,E2 8548.019} C_VEL
LIN {X 0,Y 436.942,Z 763.68,A -85,B 0,C 180,E1 8551.99,E2 8551.99} C_VEL
LIN {X 0,Y 437.016,Z 758.612,A -85,B 0,C 180,E1 8555.971,E2 8555.971} C_VEL
LIN {X 0,Y 437.026,Z 748.197,A -85,B 0,C 180,E1 8559.98,E2 8559.98} C_VEL
LIN {X 0,Y 437.63,Z 731.827,A -85,B 0,C 180,E1 8564.02,E2 8564.02} C_VEL
LIN {X 0,Y 438.877,Z 709.379,A -85,B 0,C 180,E1 8567.834,E2 8567.834} C_VEL
LIN {X 0,Y 440.885,Z 683.195,A -85,B 0,C 180,E1 8571.009,E2 8571.009} C_VEL
LIN {X 0,Y 443.217,Z 652.705,A -85,B 0,C 180,E1 8573.633,E2 8573.633} C_VEL
LIN {X 0,Y 445.564,Z 619.072,A -85,B 0,C 180,E1 8575.55,E2 8575.55} C_VEL
LIN {X 0,Y 447.049,Z 584.069,A -85,B 0,C 180,E1 8576.686,E2 8576.686} C_VEL
LIN {X 0,Y 446.497,Z 562.747,A -85,B 0,C 180,E1 8577.129,E2 8577.129} C_VEL
LIN {X 0,Y 437.839,Z 534.632,A -85,B 0,C 180,E1 8578.221,E2 8578.221} C_VEL
LIN {X 0,Y 435.174,Z 526.81,A -85,B 0,C 180,E1 8578.617,E2 8578.617} C_VEL
LIN {X 0,Y 434.998,Z 526.81,A -85,B 0,C 180,E1 8583.847,E2 8583.847} C_VEL
LIN {X 0,Y 434.947,Z 526.81,A -85,B 0,C 180,E1 8590.032,E2 8590.032} C_VEL
LIN {X 0,Y 434.998,Z 526.81,A -85,B 0,C 180,E1 8595.894,E2 8595.894} C_VEL
LIN {X 0,Y 434.91,Z 526.81,A -85,B 0,C 180,E1 8601.208,E2 8601.208} C_VEL
LIN {X 0,Y 435.1,Z 526.81,A -85,B 0,C 180,E1 8606.641,E2 8606.641} C_VEL
LIN {X 0,Y 435.17,Z 526.81,A -85,B 0,C 180,E1 8613.117,E2 8613.117} C_VEL
LIN {X 0,Y 435.385,Z 526.81,A -85,B 0,C 180,E1 8619.887,E2 8619.887} C_VEL
LIN {X 0,Y 435.44,Z 527.511,A -85,B 0,C 180,E1 8621.771,E2 8621.771} C_VEL
LIN {X 0,Y 442.625,Z 554.075,A -85,B 0,C 180,E1 8623.414,E2 8623.414} C_VEL
LIN {X 0,Y 442.161,Z 579.327,A -85,B 0,C 180,E1 8625.253,E2 8625.253} C_VEL
LIN {X 0,Y 440.651,Z 601.008,A -85,B 0,C 180,E1 8627.606,E2 8627.606} C_VEL
LIN {X 0,Y 439.318,Z 617.848,A -85,B 0,C 180,E1 8630.334,E2 8630.334} C_VEL
LIN {X 0,Y 438.374,Z 630.309,A -85,B 0,C 180,E1 8633.561,E2 8633.561} C_VEL
LIN {X 0,Y 437.852,Z 637.22,A -85,B 0,C 180,E1 8637.033,E2 8637.033} C_VEL
LIN {X 0,Y 437.559,Z 638.488,A -85,B 0,C 180,E1 8640.006,E2 8640.006} C_VEL
LIN {X 0,Y 437.591,Z 635.574,A -85,B 0,C 180,E1 8642.981,E2 8642.981} C_VEL
LIN {X 0,Y 437.897,Z 626.645,A -85,B 0,C 180,E1 8646.458,E2 8646.458} C_VEL
LIN {X 0,Y 438.614,Z 611.954,A -85,B 0,C 180,E1 8649.694,E2 8649.694} C_VEL
LIN {X 0,Y 439.677,Z 592.656,A -85,B 0,C 180,E1 8652.434,E2 8652.434} C_VEL
LIN {X 0,Y 440.856,Z 569.411,A -85,B 0,C 180,E1 8654.622,E2 8654.622} C_VEL
LIN {X 0,Y 440.648,Z 551.358,A -85,B 0,C 180,E1 8655.812,E2 8655.812} C_VEL
LIN {X 0,Y 435.506,Z 526.81,A -85,B 0,C 180,E1 8657.087,E2 8657.087} C_VEL
LIN {X 0,Y 435.344,Z 526.81,A -85,B 0,C 180,E1 8662.498,E2 8662.498} C_VEL
LIN {X 0,Y 435.053,Z 526.81,A -85,B 0,C 180,E1 8669.526,E2 8669.526} C_VEL
LIN {X 0,Y 435.005,Z 526.81,A -85,B 0,C 180,E1 8673.847,E2 8673.847} C_VEL
LIN {X 0,Y 434.87,Z 526.81,A -85,B 0,C 180,E1 8680,E2 8680} C_VEL
LIN {X 0,Y 434.954,Z 526.81,A -85,B 0,C 180,E1 8686.977,E2 8686.977} C_VEL
LIN {X 0,Y 434.958,Z 526.81,A -85,B 0,C 180,E1 8693.712,E2 8693.712} C_VEL
LIN {X 0,Y 435.065,Z 526.81,A -85,B 0,C 180,E1 8698.527,E2 8698.527} C_VEL
LIN {X 0,Y 435.263,Z 526.81,A -85,B 0,C 180,E1 8705.323,E2 8705.323} C_VEL
LIN {X 0,Y 435.472,Z 526.81,A -85,B 0,C 180,E1 8711.76,E2 8711.76} C_VEL
LIN {X 0,Y 435.519,Z 526.81,A -85,B 0,C 180,E1 8717.956,E2 8717.956} C_VEL
LIN {X 0,Y 435.881,Z 526.81,A -85,B 0,C 180,E1 8724.014,E2 8724.014} C_VEL
LIN {X 0,Y 436.156,Z 526.81,A -85,B 0,C 180,E1 8729.995,E2 8729.995} C_VEL
LIN {X 0,Y 435.845,Z 526.81,A -85,B 0,C 180,E1 8735.977,E2 8735.977} C_VEL
LIN {X 0,Y 435.617,Z 526.81,A -85,B 0,C 180,E1 8742.032,E2 8742.032} C_VEL
LIN {X 0,Y 435.473,Z 526.81,A -85,B 0,C 180,E1 8748.23,E2 8748.23} C_VEL
LIN {X 0,Y 435.181,Z 526.81,A -85,B 0,C 180,E1 8755.225,E2 8755.225} C_VEL
LIN {X 0,Y 435.043,Z 526.81,A -85,B 0,C 180,E1 8761.464,E2 8761.464} C_VEL
LIN {X 0,Y 434.88,Z 526.81,A -85,B 0,C 180,E1 8766.791,E2 8766.791} C_VEL
LIN {X 0,Y 434.867,Z 526.81,A -85,B 0,C 180,E1 8773.011,E2 8773.011} C_VEL
LIN {X 0,Y 434.967,Z 526.81,A -85,B 0,C 180,E1 8778.59,E2 8778.59} C_VEL
LIN {X 0,Y 434.936,Z 526.81,A -85,B 0,C 180,E1 8783.71,E2 8783.71} C_VEL
LIN {X 0,Y 435.056,Z 526.81,A -85,B 0,C 180,E1 8788.526,E2 8788.526} C_VEL
LIN {X 0,Y 435.25,Z 526.81,A -85,B 0,C 180,E1 8795.322,E2 8795.322} C_VEL
LIN {X 0,Y 435.489,Z 526.81,A -85,B 0,C 180,E1 8801.76,E2 8801.76} C_VEL
LIN {X 0,Y 435.517,Z 526.81,A -85,B 0,C 180,E1 8807.955,E2 8807.955} C_VEL
LIN {X 0,Y 435.896,Z 526.81,A -85,B 0,C 180,E1 8814.013,E2 8814.013} C_VEL
LIN {X 0,Y 436.122,Z 526.81,A -85,B 0,C 180,E1 8819.994,E2 8819.994} C_VEL
LIN {X 0,Y 435.806,Z 526.81,A -85,B 0,C 180,E1 8825.976,E2 8825.976} C_VEL
LIN {X 0,Y 435.563,Z 526.81,A -85,B 0,C 180,E1 8832.031,E2 8832.031} C_VEL
LIN {X 0,Y 435.427,Z 526.81,A -85,B 0,C 180,E1 8838.23,E2 8838.23} C_VEL
LIN {X 0,Y 435.176,Z 526.81,A -85,B 0,C 180,E1 8845.242,E2 8845.242} C_VEL
LIN {X 0,Y 435.091,Z 526.81,A -85,B 0,C 180,E1 8851.456,E2 8851.456} C_VEL
LIN {X 0,Y 434.963,Z 526.81,A -85,B 0,C 180,E1 8856.82,E2 8856.82} C_VEL
LIN {X 0,Y 434.798,Z 526.81,A -85,B 0,C 180,E1 8863.014,E2 8863.014} C_VEL
LIN {X 0,Y 434.778,Z 526.81,A -85,B 0,C 180,E1 8869.994,E2 8869.994} C_VEL
LIN {X 0,Y 434.995,Z 526.81,A -85,B 0,C 180,E1 8876.637,E2 8876.637} C_VEL
LIN {X 0,Y 435.231,Z 526.81,A -85,B 0,C 180,E1 8881.633,E2 8881.633} C_VEL
LIN {X 0,Y 447.443,Z 568.759,A -85,B 0,C 180,E1 8883.012,E2 8883.012} C_VEL
LIN {X 0,Y 446.492,Z 607.688,A -85,B 0,C 180,E1 8883.899,E2 8883.899} C_VEL
LIN {X 0,Y 445.296,Z 628.247,A -85,B 0,C 180,E1 8884.75,E2 8884.75} C_VEL
LIN {X 0,Y 440.358,Z 644.273,A -85,B 0,C 180,E1 8885.495,E2 8885.495} C_VEL
LIN {X 0,Y 435.37,Z 659.358,A -85,B 0,C 180,E1 8886.411,E2 8886.411} C_VEL
LIN {X 0,Y 432.961,Z 688.619,A -85,B 0,C 180,E1 8889.135,E2 8889.135} C_VEL
LIN {X 0,Y 430.942,Z 713.25,A -85,B 0,C 180,E1 8892.365,E2 8892.365} C_VEL
LIN {X 0,Y 429.646,Z 734.325,A -85,B 0,C 180,E1 8896.244,E2 8896.244} C_VEL
LIN {X 0,Y 429.085,Z 749.16,A -85,B 0,C 180,E1 8900.218,E2 8900.218} C_VEL
LIN {X 0,Y 429.099,Z 758.051,A -85,B 0,C 180,E1 8903.928,E2 8903.928} C_VEL
LIN {X 0,Y 429.129,Z 762.76,A -85,B 0,C 180,E1 8907.983,E2 8907.983} C_VEL
LIN {X 0,Y 429.117,Z 762.552,A -85,B 0,C 180,E1 8912.027,E2 8912.027} C_VEL
LIN {X 0,Y 429.189,Z 757.447,A -85,B 0,C 180,E1 8916.08,E2 8916.08} C_VEL
LIN {X 0,Y 429.17,Z 746.964,A -85,B 0,C 180,E1 8920.165,E2 8920.165} C_VEL
LIN {X 0,Y 429.8,Z 730.513,A -85,B 0,C 180,E1 8924.281,E2 8924.281} C_VEL
LIN {X 0,Y 431.184,Z 707.99,A -85,B 0,C 180,E1 8928.163,E2 8928.163} C_VEL
LIN {X 0,Y 433.388,Z 680.478,A -85,B 0,C 180,E1 8931.525,E2 8931.525} C_VEL
LIN {X 0,Y 435.759,Z 650.579,A -85,B 0,C 180,E1 8934.101,E2 8934.101} C_VEL
LIN {X 0,Y 438.29,Z 617.177,A -85,B 0,C 180,E1 8936.009,E2 8936.009} C_VEL
LIN {X 0,Y 439.919,Z 581.632,A -85,B 0,C 180,E1 8937.154,E2 8937.154} C_VEL
LIN {X 0,Y 439.335,Z 564.168,A -85,B 0,C 180,E1 8937.539,E2 8937.539} C_VEL
LIN {X 0,Y 431.152,Z 537.707,A -85,B 0,C 180,E1 8938.626,E2 8938.626} C_VEL
LIN {X 0,Y 427.155,Z 526.81,A -85,B 0,C 180,E1 8939.237,E2 8939.237} C_VEL
LIN {X 0,Y 426.959,Z 526.81,A -85,B 0,C 180,E1 8945.366,E2 8945.366} C_VEL
LIN {X 0,Y 427.066,Z 526.81,A -85,B 0,C 180,E1 8951.896,E2 8951.896} C_VEL
LIN {X 0,Y 427.012,Z 526.81,A -85,B 0,C 180,E1 8958.132,E2 8958.132} C_VEL
LIN {X 0,Y 427.002,Z 526.81,A -85,B 0,C 180,E1 8964.649,E2 8964.649} C_VEL
LIN {X 0,Y 427.179,Z 526.81,A -85,B 0,C 180,E1 8970.26,E2 8970.26} C_VEL
LIN {X 0,Y 427.313,Z 526.81,A -85,B 0,C 180,E1 8977.12,E2 8977.12} C_VEL
LIN {X 0,Y 427.481,Z 527.113,A -85,B 0,C 180,E1 8981.193,E2 8981.193} C_VEL
LIN {X 0,Y 435.141,Z 554.66,A -85,B 0,C 180,E1 8982.977,E2 8982.977} C_VEL
LIN {X 0,Y 435.423,Z 570.795,A -85,B 0,C 180,E1 8984.115,E2 8984.115} C_VEL
LIN {X 0,Y 433.771,Z 594.803,A -85,B 0,C 180,E1 8986.38,E2 8986.38} C_VEL
LIN {X 0,Y 432.093,Z 614.423,A -85,B 0,C 180,E1 8989.214,E2 8989.214} C_VEL
LIN {X 0,Y 431.001,Z 628.61,A -85,B 0,C 180,E1 8992.437,E2 8992.437} C_VEL
LIN {X 0,Y 430.24,Z 637.212,A -85,B 0,C 180,E1 8995.97,E2 8995.97} C_VEL
LIN {X 0,Y 429.921,Z 639.349,A -85,B 0,C 180,E1 8997.988,E2 8997.988} C_VEL
LIN {X 0,Y 429.749,Z 639.671,A -85,B 0,C 180,E1 9000.006,E2 9000.006} C_VEL
LIN {X 0,Y 429.772,Z 636.641,A -85,B 0,C 180,E1 9003.035,E2 9003.035} C_VEL
LIN {X 0,Y 430.099,Z 627.532,A -85,B 0,C 180,E1 9006.575,E2 9006.575} C_VEL
LIN {X 0,Y 430.853,Z 612.619,A -85,B 0,C 180,E1 9009.87,E2 9009.87} C_VEL
LIN {X 0,Y 431.958,Z 593.076,A -85,B 0,C 180,E1 9012.66,E2 9012.66} C_VEL
LIN {X 0,Y 433.267,Z 568.99,A -85,B 0,C 180,E1 9014.927,E2 9014.927} C_VEL
LIN {X 0,Y 432.922,Z 552.348,A -85,B 0,C 180,E1 9016.04,E2 9016.04} C_VEL
LIN {X 0,Y 427.576,Z 526.81,A -85,B 0,C 180,E1 9017.39,E2 9017.39} C_VEL
LIN {X 0,Y 427.395,Z 526.81,A -85,B 0,C 180,E1 9022.94,E2 9022.94} C_VEL
LIN {X 0,Y 427.158,Z 526.81,A -85,B 0,C 180,E1 9029.757,E2 9029.757} C_VEL
LIN {X 0,Y 426.965,Z 526.81,A -85,B 0,C 180,E1 9037.079,E2 9037.079} C_VEL
LIN {X 0,Y 426.958,Z 526.81,A -85,B 0,C 180,E1 9042.365,E2 9042.365} C_VEL
LIN {X 0,Y 427.042,Z 526.81,A -85,B 0,C 180,E1 9048.127,E2 9048.127} C_VEL
LIN {X 0,Y 427.002,Z 526.81,A -85,B 0,C 180,E1 9054.647,E2 9054.647} C_VEL
LIN {X 0,Y 427.175,Z 526.81,A -85,B 0,C 180,E1 9060.245,E2 9060.245} C_VEL
LIN {X 0,Y 427.39,Z 526.81,A -85,B 0,C 180,E1 9067.093,E2 9067.093} C_VEL
LIN {X 0,Y 427.521,Z 526.81,A -85,B 0,C 180,E1 9073.537,E2 9073.537} C_VEL
LIN {X 0,Y 427.688,Z 526.81,A -85,B 0,C 180,E1 9079.8,E2 9079.8} C_VEL
LIN {X 0,Y 427.984,Z 526.81,A -85,B 0,C 180,E1 9085.938,E2 9085.938} C_VEL
LIN {X 0,Y 428.13,Z 526.81,A -85,B 0,C 180,E1 9092.022,E2 9092.022} C_VEL
LIN {X 0,Y 427.9,Z 526.81,A -85,B 0,C 180,E1 9098.132,E2 9098.132} C_VEL
LIN {X 0,Y 427.638,Z 526.81,A -85,B 0,C 180,E1 9104.345,E2 9104.345} C_VEL
LIN {X 0,Y 427.439,Z 526.81,A -85,B 0,C 180,E1 9110.74,E2 9110.74} C_VEL
LIN {X 0,Y 427.185,Z 526.81,A -85,B 0,C 180,E1 9117.608,E2 9117.608} C_VEL
LIN {X 0,Y 427.097,Z 526.81,A -85,B 0,C 180,E1 9122.118,E2 9122.118} C_VEL
LIN {X 0,Y 426.959,Z 526.81,A -85,B 0,C 180,E1 9128.719,E2 9128.719} C_VEL
LIN {X 0,Y 427.001,Z 526.81,A -85,B 0,C 180,E1 9135.16,E2 9135.16} C_VEL
LIN {X 0,Y 427.03,Z 526.81,A -85,B 0,C 180,E1 9141.255,E2 9141.255} C_VEL
LIN {X 0,Y 427.146,Z 526.81,A -85,B 0,C 180,E1 9148.279,E2 9148.279} C_VEL
LIN {X 0,Y 427.323,Z 526.81,A -85,B 0,C 180,E1 9154.833,E2 9154.833} C_VEL
LIN {X 0,Y 427.571,Z 526.81,A -85,B 0,C 180,E1 9161.41,E2 9161.41} C_VEL
LIN {X 0,Y 427.595,Z 526.81,A -85,B 0,C 180,E1 9167.728,E2 9167.728} C_VEL
LIN {X 0,Y 427.977,Z 526.81,A -85,B 0,C 180,E1 9173.902,E2 9173.902} C_VEL
LIN {X 0,Y 428.221,Z 526.81,A -85,B 0,C 180,E1 9179.994,E2 9179.994} C_VEL
LIN {X 0,Y 427.889,Z 526.81,A -85,B 0,C 180,E1 9186.087,E2 9186.087} C_VEL
LIN {X 0,Y 427.64,Z 526.81,A -85,B 0,C 180,E1 9192.258,E2 9192.258} C_VEL
LIN {X 0,Y 427.508,Z 526.81,A -85,B 0,C 180,E1 9198.579,E2 9198.579} C_VEL
LIN {X 0,Y 427.291,Z 526.81,A -85,B 0,C 180,E1 9205.156,E2 9205.156} C_VEL
LIN {X 0,Y 427.177,Z 526.81,A -85,B 0,C 180,E1 9212.108,E2 9212.108} C_VEL
LIN {X 0,Y 427.005,Z 526.81,A -85,B 0,C 180,E1 9218.741,E2 9218.741} C_VEL
LIN {X 0,Y 426.847,Z 526.81,A -85,B 0,C 180,E1 9225.176,E2 9225.176} C_VEL
LIN {X 0,Y 426.898,Z 526.81,A -85,B 0,C 180,E1 9231.271,E2 9231.271} C_VEL
LIN {X 0,Y 427.105,Z 526.81,A -85,B 0,C 180,E1 9238.281,E2 9238.281} C_VEL
LIN {X 0,Y 427.289,Z 526.81,A -85,B 0,C 180,E1 9241.27,E2 9241.27} C_VEL
LIN {X 0,Y 440.007,Z 569.839,A -85,B 0,C 180,E1 9242.691,E2 9242.691} C_VEL
LIN {X 0,Y 438.936,Z 608.31,A -85,B 0,C 180,E1 9243.609,E2 9243.609} C_VEL
LIN {X 0,Y 436.782,Z 641.897,A -85,B 0,C 180,E1 9245.212,E2 9245.212} C_VEL
LIN {X 0,Y 435.37,Z 659.358,A -85,B 0,C 180,E1 9246.411,E2 9246.411} C_VEL
LIN {X 0,Y 430.331,Z 673.948,A -85,B 0,C 180,E1 9247.539,E2 9247.539} C_VEL
LIN {X 0,Y 425.269,Z 687.547,A -85,B 0,C 180,E1 9248.846,E2 9248.846} C_VEL
LIN {X 0,Y 423.087,Z 713.294,A -85,B 0,C 180,E1 9252.296,E2 9252.296} C_VEL
LIN {X 0,Y 421.813,Z 733.574,A -85,B 0,C 180,E1 9256.135,E2 9256.135} C_VEL
LIN {X 0,Y 421.212,Z 748.614,A -85,B 0,C 180,E1 9260.273,E2 9260.273} C_VEL
LIN {X 0,Y 421.249,Z 756.866,A -85,B 0,C 180,E1 9263.815,E2 9263.815} C_VEL
LIN {X 0,Y 421.319,Z 761.633,A -85,B 0,C 180,E1 9267.945,E2 9267.945} C_VEL
LIN {X 0,Y 421.309,Z 761.423,A -85,B 0,C 180,E1 9272.064,E2 9272.064} C_VEL
LIN {X 0,Y 421.33,Z 756.281,A -85,B 0,C 180,E1 9276.194,E2 9276.194} C_VEL
LIN {X 0,Y 421.312,Z 745.747,A -85,B 0,C 180,E1 9280.356,E2 9280.356} C_VEL
LIN {X 0,Y 421.98,Z 729.23,A -85,B 0,C 180,E1 9284.551,E2 9284.551} C_VEL
LIN {X 0,Y 423.473,Z 706.647,A -85,B 0,C 180,E1 9288.506,E2 9288.506} C_VEL
LIN {X 0,Y 425.755,Z 679.638,A -85,B 0,C 180,E1 9291.867,E2 9291.867} C_VEL
LIN {X 0,Y 428.37,Z 649.114,A -85,B 0,C 180,E1 9294.544,E2 9294.544} C_VEL
LIN {X 0,Y 431.078,Z 615.627,A -85,B 0,C 180,E1 9296.477,E2 9296.477} C_VEL
LIN {X 0,Y 432.81,Z 579.953,A -85,B 0,C 180,E1 9297.635,E2 9297.635} C_VEL
LIN {X 0,Y 432.263,Z 565.574,A -85,B 0,C 180,E1 9297.973,E2 9297.973} C_VEL
LIN {X 0,Y 423.627,Z 538.337,A -85,B 0,C 180,E1 9299.178,E2 9299.178} C_VEL
LIN {X 0,Y 419.242,Z 526.81,A -85,B 0,C 180,E1 9299.935,E2 9299.935} C_VEL
LIN {X 0,Y 419.077,Z 526.81,A -85,B 0,C 180,E1 9307.375,E2 9307.375} C_VEL
LIN {X 0,Y 419.062,Z 526.81,A -85,B 0,C 180,E1 9313.743,E2 9313.743} C_VEL
LIN {X 0,Y 419.038,Z 526.81,A -85,B 0,C 180,E1 9319.441,E2 9319.441} C_VEL
LIN {X 0,Y 419.114,Z 526.81,A -85,B 0,C 180,E1 9326.198,E2 9326.198} C_VEL
LIN {X 0,Y 419.26,Z 526.81,A -85,B 0,C 180,E1 9332.009,E2 9332.009} C_VEL
LIN {X 0,Y 419.428,Z 526.81,A -85,B 0,C 180,E1 9338.847,E2 9338.847} C_VEL
LIN {X 0,Y 419.594,Z 526.937,A -85,B 0,C 180,E1 9340.583,E2 9340.583} C_VEL
LIN {X 0,Y 427.673,Z 554.94,A -85,B 0,C 180,E1 9342.496,E2 9342.496} C_VEL
LIN {X 0,Y 428.353,Z 569.919,A -85,B 0,C 180,E1 9343.582,E2 9343.582} C_VEL
LIN {X 0,Y 426.485,Z 594.508,A -85,B 0,C 180,E1 9345.88,E2 9345.88} C_VEL
LIN {X 0,Y 424.652,Z 614.679,A -85,B 0,C 180,E1 9348.758,E2 9348.758} C_VEL
LIN {X 0,Y 423.425,Z 628.346,A -85,B 0,C 180,E1 9351.784,E2 9351.784} C_VEL
LIN {X 0,Y 422.654,Z 636.779,A -85,B 0,C 180,E1 9354.868,E2 9354.868} C_VEL
LIN {X 0,Y 422.151,Z 640.625,A -85,B 0,C 180,E1 9357.951,E2 9357.951} C_VEL
LIN {X 0,Y 421.96,Z 640.854,A -85,B 0,C 180,E1 9360.006,E2 9360.006} C_VEL
LIN {X 0,Y 421.953,Z 636.742,A -85,B 0,C 180,E1 9363.606,E2 9363.606} C_VEL
LIN {X 0,Y 422.41,Z 626.54,A -85,B 0,C 180,E1 9367.213,E2 9367.213} C_VEL
LIN {X 0,Y 423.205,Z 611.845,A -85,B 0,C 180,E1 9370.31,E2 9370.31} C_VEL
LIN {X 0,Y 424.427,Z 591.256,A -85,B 0,C 180,E1 9373.151,E2 9373.151} C_VEL
LIN {X 0,Y 425.742,Z 566.478,A -85,B 0,C 180,E1 9375.393,E2 9375.393} C_VEL
LIN {X 0,Y 425.303,Z 553.724,A -85,B 0,C 180,E1 9376.251,E2 9376.251} C_VEL
LIN {X 0,Y 419.673,Z 526.81,A -85,B 0,C 180,E1 9377.757,E2 9377.757} C_VEL
LIN {X 0,Y 419.428,Z 526.81,A -85,B 0,C 180,E1 9383.402,E2 9383.402} C_VEL
LIN {X 0,Y 419.224,Z 526.81,A -85,B 0,C 180,E1 9390.378,E2 9390.378} C_VEL
LIN {X 0,Y 419.07,Z 526.81,A -85,B 0,C 180,E1 9397.352,E2 9397.352} C_VEL
LIN {X 0,Y 418.991,Z 526.81,A -85,B 0,C 180,E1 9403.713,E2 9403.713} C_VEL
LIN {X 0,Y 419.069,Z 526.81,A -85,B 0,C 180,E1 9409.427,E2 9409.427} C_VEL
LIN {X 0,Y 419.096,Z 526.81,A -85,B 0,C 180,E1 9416.2,E2 9416.2} C_VEL
LIN {X 0,Y 419.287,Z 526.81,A -85,B 0,C 180,E1 9421.997,E2 9421.997} C_VEL
LIN {X 0,Y 419.536,Z 526.81,A -85,B 0,C 180,E1 9428.84,E2 9428.84} C_VEL
LIN {X 0,Y 419.596,Z 526.81,A -85,B 0,C 180,E1 9435.364,E2 9435.364} C_VEL
LIN {X 0,Y 419.963,Z 526.81,A -85,B 0,C 180,E1 9441.704,E2 9441.704} C_VEL
LIN {X 0,Y 420.345,Z 526.81,A -85,B 0,C 180,E1 9447.931,E2 9447.931} C_VEL
LIN {X 0,Y 420.221,Z 526.81,A -85,B 0,C 180,E1 9454.127,E2 9454.127} C_VEL
LIN {X 0,Y 419.871,Z 526.81,A -85,B 0,C 180,E1 9460.382,E2 9460.382} C_VEL
LIN {X 0,Y 419.709,Z 526.81,A -85,B 0,C 180,E1 9466.769,E2 9466.769} C_VEL
LIN {X 0,Y 419.396,Z 526.81,A -85,B 0,C 180,E1 9473.392,E2 9473.392} C_VEL
LIN {X 0,Y 419.197,Z 526.81,A -85,B 0,C 180,E1 9480.369,E2 9480.369} C_VEL
LIN {X 0,Y 419.048,Z 526.81,A -85,B 0,C 180,E1 9487.349,E2 9487.349} C_VEL
LIN {X 0,Y 418.972,Z 526.81,A -85,B 0,C 180,E1 9493.712,E2 9493.712} C_VEL
LIN {X 0,Y 419.055,Z 526.81,A -85,B 0,C 180,E1 9499.426,E2 9499.426} C_VEL
LIN {X 0,Y 419.076,Z 526.81,A -85,B 0,C 180,E1 9506.189,E2 9506.189} C_VEL
LIN {X 0,Y 419.262,Z 526.81,A -85,B 0,C 180,E1 9511.995,E2 9511.995} C_VEL
LIN {X 0,Y 419.546,Z 526.81,A -85,B 0,C 180,E1 9518.84,E2 9518.84} C_VEL
LIN {X 0,Y 419.639,Z 526.81,A -85,B 0,C 180,E1 9525.365,E2 9525.365} C_VEL
LIN {X 0,Y 419.946,Z 526.81,A -85,B 0,C 180,E1 9531.702,E2 9531.702} C_VEL
LIN {X 0,Y 420.313,Z 526.81,A -85,B 0,C 180,E1 9537.929,E2 9537.929} C_VEL
LIN {X 0,Y 420.182,Z 526.81,A -85,B 0,C 180,E1 9544.126,E2 9544.126} C_VEL
LIN {X 0,Y 419.815,Z 526.81,A -85,B 0,C 180,E1 9550.382,E2 9550.382} C_VEL
LIN {X 0,Y 419.66,Z 526.81,A -85,B 0,C 180,E1 9556.768,E2 9556.768} C_VEL
LIN {X 0,Y 419.382,Z 526.81,A -85,B 0,C 180,E1 9563.39,E2 9563.39} C_VEL
LIN {X 0,Y 419.23,Z 526.81,A -85,B 0,C 180,E1 9570.363,E2 9570.363} C_VEL
LIN {X 0,Y 419.102,Z 526.81,A -85,B 0,C 180,E1 9577.373,E2 9577.373} C_VEL
LIN {X 0,Y 418.871,Z 526.81,A -85,B 0,C 180,E1 9583.71,E2 9583.71} C_VEL
LIN {X 0,Y 418.898,Z 526.81,A -85,B 0,C 180,E1 9589.42,E2 9589.42} C_VEL
LIN {X 0,Y 419.016,Z 526.81,A -85,B 0,C 180,E1 9596.194,E2 9596.194} C_VEL
LIN {X 0,Y 419.335,Z 527.258,A -85,B 0,C 180,E1 9600.896,E2 9600.896} C_VEL
LIN {X 0,Y 432.447,Z 569.27,A -85,B 0,C 180,E1 9602.33,E2 9602.33} C_VEL
LIN {X 0,Y 431.449,Z 607.606,A -85,B 0,C 180,E1 9603.267,E2 9603.267} C_VEL
LIN {X 0,Y 429.243,Z 640.673,A -85,B 0,C 180,E1 9604.866,E2 9604.866} C_VEL
LIN {X 0,Y 426.732,Z 671.041,A -85,B 0,C 180,E1 9607.173,E2 9607.173} C_VEL
LIN {X 0,Y 425.269,Z 687.547,A -85,B 0,C 180,E1 9608.846,E2 9608.846} C_VEL
LIN {X 0,Y 420.169,Z 700.263,A -85,B 0,C 180,E1 9610.333,E2 9610.333} C_VEL
LIN {X 0,Y 415.304,Z 711.905,A -85,B 0,C 180,E1 9612.008,E2 9612.008} C_VEL
LIN {X 0,Y 413.954,Z 732.643,A -85,B 0,C 180,E1 9615.989,E2 9615.989} C_VEL
LIN {X 0,Y 413.376,Z 747.015,A -85,B 0,C 180,E1 9619.986,E2 9619.986} C_VEL
LIN {X 0,Y 413.428,Z 755.651,A -85,B 0,C 180,E1 9623.697,E2 9623.697} C_VEL
LIN {X 0,Y 413.493,Z 760.486,A -85,B 0,C 180,E1 9627.907,E2 9627.907} C_VEL
LIN {X 0,Y 413.483,Z 760.288,A -85,B 0,C 180,E1 9632.103,E2 9632.103} C_VEL
LIN {X 0,Y 413.504,Z 755.124,A -85,B 0,C 180,E1 9636.311,E2 9636.311} C_VEL
LIN {X 0,Y 413.459,Z 744.549,A -85,B 0,C 180,E1 9640.555,E2 9640.555} C_VEL
LIN {X 0,Y 414.141,Z 727.977,A -85,B 0,C 180,E1 9644.833,E2 9644.833} C_VEL
LIN {X 0,Y 415.766,Z 705.268,A -85,B 0,C 180,E1 9648.876,E2 9648.876} C_VEL
LIN {X 0,Y 418.207,Z 678.258,A -85,B 0,C 180,E1 9652.29,E2 9652.29} C_VEL
LIN {X 0,Y 421.041,Z 647.807,A -85,B 0,C 180,E1 9655,E2 9655} C_VEL
LIN {X 0,Y 423.962,Z 614.054,A -85,B 0,C 180,E1 9656.973,E2 9656.973} C_VEL
LIN {X 0,Y 425.737,Z 580.379,A -85,B 0,C 180,E1 9658.099,E2 9658.099} C_VEL
LIN {X 0,Y 425.231,Z 567.032,A -85,B 0,C 180,E1 9658.432,E2 9658.432} C_VEL
LIN {X 0,Y 416.733,Z 540.564,A -85,B 0,C 180,E1 9659.684,E2 9659.684} C_VEL
LIN {X 0,Y 411.252,Z 526.81,A -85,B 0,C 180,E1 9660.564,E2 9660.564} C_VEL
LIN {X 0,Y 411.133,Z 526.81,A -85,B 0,C 180,E1 9666.108,E2 9666.108} C_VEL
LIN {X 0,Y 411.093,Z 526.81,A -85,B 0,C 180,E1 9672.57,E2 9672.57} C_VEL
LIN {X 0,Y 411.052,Z 526.81,A -85,B 0,C 180,E1 9678.481,E2 9678.481} C_VEL
LIN {X 0,Y 411.174,Z 526.81,A -85,B 0,C 180,E1 9684.115,E2 9684.115} C_VEL
LIN {X 0,Y 411.336,Z 526.81,A -85,B 0,C 180,E1 9691.421,E2 9691.421} C_VEL
LIN {X 0,Y 411.466,Z 526.81,A -85,B 0,C 180,E1 9698.418,E2 9698.418} C_VEL
LIN {X 0,Y 411.652,Z 526.995,A -85,B 0,C 180,E1 9699.923,E2 9699.923} C_VEL
LIN {X 0,Y 420.302,Z 555.452,A -85,B 0,C 180,E1 9701.99,E2 9701.99} C_VEL
LIN {X 0,Y 421.21,Z 570.438,A -85,B 0,C 180,E1 9703.126,E2 9703.126} C_VEL
LIN {X 0,Y 419.169,Z 595.514,A -85,B 0,C 180,E1 9705.495,E2 9705.495} C_VEL
LIN {X 0,Y 417.255,Z 614.967,A -85,B 0,C 180,E1 9708.289,E2 9708.289} C_VEL
LIN {X 0,Y 415.769,Z 629.922,A -85,B 0,C 180,E1 9711.631,E2 9711.631} C_VEL
LIN {X 0,Y 414.938,Z 638.194,A -85,B 0,C 180,E1 9714.773,E2 9714.773} C_VEL
LIN {X 0,Y 414.372,Z 641.905,A -85,B 0,C 180,E1 9717.913,E2 9717.913} C_VEL
LIN {X 0,Y 414.175,Z 642.037,A -85,B 0,C 180,E1 9720.006,E2 9720.006} C_VEL
LIN {X 0,Y 414.132,Z 637.759,A -85,B 0,C 180,E1 9723.675,E2 9723.675} C_VEL
LIN {X 0,Y 414.612,Z 627.342,A -85,B 0,C 180,E1 9727.349,E2 9727.349} C_VEL
LIN {X 0,Y 415.454,Z 612.439,A -85,B 0,C 180,E1 9730.505,E2 9730.505} C_VEL
LIN {X 0,Y 416.731,Z 591.616,A -85,B 0,C 180,E1 9733.398,E2 9733.398} C_VEL
LIN {X 0,Y 418.14,Z 566.181,A -85,B 0,C 180,E1 9735.708,E2 9735.708} C_VEL
LIN {X 0,Y 417.355,Z 553.561,A -85,B 0,C 180,E1 9736.566,E2 9736.566} C_VEL
LIN {X 0,Y 411.755,Z 526.81,A -85,B 0,C 180,E1 9738.015,E2 9738.015} C_VEL
LIN {X 0,Y 411.475,Z 526.81,A -85,B 0,C 180,E1 9743.882,E2 9743.882} C_VEL
LIN {X 0,Y 411.33,Z 526.81,A -85,B 0,C 180,E1 9748.594,E2 9748.594} C_VEL
LIN {X 0,Y 411.127,Z 526.81,A -85,B 0,C 180,E1 9755.876,E2 9755.876} C_VEL
LIN {X 0,Y 411.016,Z 526.81,A -85,B 0,C 180,E1 9762.538,E2 9762.538} C_VEL
LIN {X 0,Y 411.072,Z 526.81,A -85,B 0,C 180,E1 9768.466,E2 9768.466} C_VEL
LIN {X 0,Y 411.166,Z 526.81,A -85,B 0,C 180,E1 9774.115,E2 9774.115} C_VEL
LIN {X 0,Y 411.356,Z 526.81,A -85,B 0,C 180,E1 9781.408,E2 9781.408} C_VEL
LIN {X 0,Y 411.565,Z 526.81,A -85,B 0,C 180,E1 9788.41,E2 9788.41} C_VEL
LIN {X 0,Y 411.665,Z 526.81,A -85,B 0,C 180,E1 9795.076,E2 9795.076} C_VEL
LIN {X 0,Y 412.048,Z 526.81,A -85,B 0,C 180,E1 9801.543,E2 9801.543} C_VEL
LIN {X 0,Y 412.431,Z 526.81,A -85,B 0,C 180,E1 9807.891,E2 9807.891} C_VEL
LIN {X 0,Y 412.301,Z 526.81,A -85,B 0,C 180,E1 9814.207,E2 9814.207} C_VEL
LIN {X 0,Y 411.934,Z 526.81,A -85,B 0,C 180,E1 9820.585,E2 9820.585} C_VEL
LIN {X 0,Y 411.762,Z 526.81,A -85,B 0,C 180,E1 9827.102,E2 9827.102} C_VEL
LIN {X 0,Y 411.443,Z 526.81,A -85,B 0,C 180,E1 9833.872,E2 9833.872} C_VEL
LIN {X 0,Y 411.317,Z 526.81,A -85,B 0,C 180,E1 9838.584,E2 9838.584} C_VEL
LIN {X 0,Y 411.12,Z 526.81,A -85,B 0,C 180,E1 9845.876,E2 9845.876} C_VEL
LIN {X 0,Y 410.994,Z 526.81,A -85,B 0,C 180,E1 9852.536,E2 9852.536} C_VEL
LIN {X 0,Y 411.057,Z 526.81,A -85,B 0,C 180,E1 9858.465,E2 9858.465} C_VEL
LIN {X 0,Y 411.141,Z 526.81,A -85,B 0,C 180,E1 9864.104,E2 9864.104} C_VEL
LIN {X 0,Y 411.333,Z 526.81,A -85,B 0,C 180,E1 9871.406,E2 9871.406} C_VEL
LIN {X 0,Y 411.571,Z 526.81,A -85,B 0,C 180,E1 9878.41,E2 9878.41} C_VEL
LIN {X 0,Y 411.709,Z 526.81,A -85,B 0,C 180,E1 9885.077,E2 9885.077} C_VEL
LIN {X 0,Y 412.026,Z 526.81,A -85,B 0,C 180,E1 9891.541,E2 9891.541} C_VEL
LIN {X 0,Y 412.4,Z 526.81,A -85,B 0,C 180,E1 9897.89,E2 9897.89} C_VEL
LIN {X 0,Y 412.263,Z 526.81,A -85,B 0,C 180,E1 9904.206,E2 9904.206} C_VEL
LIN {X 0,Y 411.878,Z 526.81,A -85,B 0,C 180,E1 9910.584,E2 9910.584} C_VEL
LIN {X 0,Y 411.728,Z 526.81,A -85,B 0,C 180,E1 9917.101,E2 9917.101} C_VEL
LIN {X 0,Y 411.425,Z 526.81,A -85,B 0,C 180,E1 9923.871,E2 9923.871} C_VEL
LIN {X 0,Y 411.327,Z 526.81,A -85,B 0,C 180,E1 9928.58,E2 9928.58} C_VEL
LIN {X 0,Y 411.204,Z 526.81,A -85,B 0,C 180,E1 9935.908,E2 9935.908} C_VEL
LIN {X 0,Y 410.936,Z 526.81,A -85,B 0,C 180,E1 9942.54,E2 9942.54} C_VEL
LIN {X 0,Y 410.898,Z 526.81,A -85,B 0,C 180,E1 9948.458,E2 9948.458} C_VEL
LIN {X 0,Y 411.055,Z 526.81,A -85,B 0,C 180,E1 9954.114,E2 9954.114} C_VEL
LIN {X 0,Y 411.415,Z 527.309,A -85,B 0,C 180,E1 9960.496,E2 9960.496} C_VEL
LIN {X 0,Y 424.973,Z 570.433,A -85,B 0,C 180,E1 9962.006,E2 9962.006} C_VEL
LIN {X 0,Y 423.879,Z 608.17,A -85,B 0,C 180,E1 9962.973,E2 9962.973} C_VEL
LIN {X 0,Y 421.572,Z 641.133,A -85,B 0,C 180,E1 9964.618,E2 9964.618} C_VEL
LIN {X 0,Y 418.926,Z 671.8,A -85,B 0,C 180,E1 9967.026,E2 9967.026} C_VEL
LIN {X 0,Y 416.42,Z 698.752,A -85,B 0,C 180,E1 9970.076,E2 9970.076} C_VEL
LIN {X 0,Y 415.304,Z 711.905,A -85,B 0,C 180,E1 9972.008,E2 9972.008} C_VEL
LIN {X 0,Y 413.622,Z 717.408,A -85,B 0,C 180,E1 9972.923,E2 9972.923} C_VEL
LIN {X 0,Y 406.204,Z 730.59,A -85,B 0,C 180,E1 9975.578,E2 9975.578} C_VEL
LIN {X 0,Y 406.091,Z 731.704,A -85,B 0,C 180,E1 9975.844,E2 9975.844} C_VEL
LIN {X 0,Y 405.522,Z 745.663,A -85,B 0,C 180,E1 9979.79,E2 9979.79} C_VEL
LIN {X 0,Y 405.606,Z 754.413,A -85,B 0,C 180,E1 9983.575,E2 9983.575} C_VEL
LIN {X 0,Y 405.69,Z 759.331,A -85,B 0,C 180,E1 9987.866,E2 9987.866} C_VEL
LIN {X 0,Y 405.682,Z 759.149,A -85,B 0,C 180,E1 9992.144,E2 9992.144} C_VEL
LIN {X 0,Y 405.654,Z 753.968,A -85,B 0,C 180,E1 9996.434,E2 9996.434} C_VEL
LIN {X 0,Y 405.602,Z 743.369,A -85,B 0,C 180,E1 10000.762,E2 10000.762} C_VEL
LIN {X 0,Y 406.314,Z 726.761,A -85,B 0,C 180,E1 10005.125,E2 10005.125} C_VEL
LIN {X 0,Y 407.997,Z 704.688,A -85,B 0,C 180,E1 10009.142,E2 10009.142} C_VEL
LIN {X 0,Y 410.515,Z 678.77,A -85,B 0,C 180,E1 10012.528,E2 10012.528} C_VEL
LIN {X 0,Y 413.58,Z 648.429,A -85,B 0,C 180,E1 10015.338,E2 10015.338} C_VEL
LIN {X 0,Y 416.661,Z 615.642,A -85,B 0,C 180,E1 10017.351,E2 10017.351} C_VEL
LIN {X 0,Y 418.738,Z 580.839,A -85,B 0,C 180,E1 10018.589,E2 10018.589} C_VEL
LIN {X 0,Y 418.115,Z 567.98,A -85,B 0,C 180,E1 10018.942,E2 10018.942} C_VEL
LIN {X 0,Y 410.035,Z 543.054,A -85,B 0,C 180,E1 10020.203,E2 10020.203} C_VEL
LIN {X 0,Y 403.254,Z 526.81,A -85,B 0,C 180,E1 10021.353,E2 10021.353} C_VEL
LIN {X 0,Y 403.098,Z 526.81,A -85,B 0,C 180,E1 10027.943,E2 10027.943} C_VEL
LIN {X 0,Y 403.193,Z 526.81,A -85,B 0,C 180,E1 10034.493,E2 10034.493} C_VEL
LIN {X 0,Y 403.121,Z 526.81,A -85,B 0,C 180,E1 10040.331,E2 10040.331} C_VEL
LIN {X 0,Y 403.25,Z 526.81,A -85,B 0,C 180,E1 10045.733,E2 10045.733} C_VEL
LIN {X 0,Y 403.341,Z 526.81,A -85,B 0,C 180,E1 10050.8,E2 10050.8} C_VEL
LIN {X 0,Y 403.528,Z 526.81,A -85,B 0,C 180,E1 10057.971,E2 10057.971} C_VEL
LIN {X 0,Y 403.691,Z 527.602,A -85,B 0,C 180,E1 10059.209,E2 10059.209} C_VEL
LIN {X 0,Y 412.606,Z 554.269,A -85,B 0,C 180,E1 10061.313,E2 10061.313} C_VEL
LIN {X 0,Y 414.224,Z 569.584,A -85,B 0,C 180,E1 10062.528,E2 10062.528} C_VEL
LIN {X 0,Y 412.102,Z 594.369,A -85,B 0,C 180,E1 10064.832,E2 10064.832} C_VEL
LIN {X 0,Y 409.952,Z 615.245,A -85,B 0,C 180,E1 10067.793,E2 10067.793} C_VEL
LIN {X 0,Y 408.35,Z 629.654,A -85,B 0,C 180,E1 10070.941,E2 10070.941} C_VEL
LIN {X 0,Y 407.225,Z 639.643,A -85,B 0,C 180,E1 10074.674,E2 10074.674} C_VEL
LIN {X 0,Y 406.602,Z 643.206,A -85,B 0,C 180,E1 10077.873,E2 10077.873} C_VEL
LIN {X 0,Y 406.372,Z 643.222,A -85,B 0,C 180,E1 10080.007,E2 10080.007} C_VEL
LIN {X 0,Y 406.318,Z 638.776,A -85,B 0,C 180,E1 10083.745,E2 10083.745} C_VEL
LIN {X 0,Y 406.819,Z 628.122,A -85,B 0,C 180,E1 10087.491,E2 10087.491} C_VEL
LIN {X 0,Y 407.703,Z 612.959,A -85,B 0,C 180,E1 10090.707,E2 10090.707} C_VEL
LIN {X 0,Y 409.028,Z 591.831,A -85,B 0,C 180,E1 10093.655,E2 10093.655} C_VEL
LIN {X 0,Y 410.531,Z 566.005,A -85,B 0,C 180,E1 10096.005,E2 10096.005} C_VEL
LIN {X 0,Y 408.699,Z 549.738,A -85,B 0,C 180,E1 10097.111,E2 10097.111} C_VEL
LIN {X 0,Y 403.87,Z 526.81,A -85,B 0,C 180,E1 10098.29,E2 10098.29} C_VEL
LIN {X 0,Y 403.491,Z 526.81,A -85,B 0,C 180,E1 10104.385,E2 10104.385} C_VEL
LIN {X 0,Y 403.288,Z 526.81,A -85,B 0,C 180,E1 10111.715,E2 10111.715} C_VEL
LIN {X 0,Y 403.07,Z 526.81,A -85,B 0,C 180,E1 10117.915,E2 10117.915} C_VEL
LIN {X 0,Y 403.144,Z 526.81,A -85,B 0,C 180,E1 10124.466,E2 10124.466} C_VEL
LIN {X 0,Y 403.15,Z 526.81,A -85,B 0,C 180,E1 10130.317,E2 10130.317} C_VEL
LIN {X 0,Y 403.246,Z 526.81,A -85,B 0,C 180,E1 10135.716,E2 10135.716} C_VEL
LIN {X 0,Y 403.353,Z 526.81,A -85,B 0,C 180,E1 10140.786,E2 10140.786} C_VEL
LIN {X 0,Y 403.619,Z 526.81,A -85,B 0,C 180,E1 10147.963,E2 10147.963} C_VEL
LIN {X 0,Y 403.737,Z 526.81,A -85,B 0,C 180,E1 10154.776,E2 10154.776} C_VEL
LIN {X 0,Y 404.106,Z 526.81,A -85,B 0,C 180,E1 10161.376,E2 10161.376} C_VEL
LIN {X 0,Y 404.537,Z 526.81,A -85,B 0,C 180,E1 10167.85,E2 10167.85} C_VEL
LIN {X 0,Y 404.381,Z 526.81,A -85,B 0,C 180,E1 10174.289,E2 10174.289} C_VEL
LIN {X 0,Y 404.001,Z 526.81,A -85,B 0,C 180,E1 10180.795,E2 10180.795} C_VEL
LIN {X 0,Y 403.804,Z 526.81,A -85,B 0,C 180,E1 10187.45,E2 10187.45} C_VEL
LIN {X 0,Y 403.461,Z 526.81,A -85,B 0,C 180,E1 10194.375,E2 10194.375} C_VEL
LIN {X 0,Y 403.269,Z 526.81,A -85,B 0,C 180,E1 10201.705,E2 10201.705} C_VEL
LIN {X 0,Y 403.047,Z 526.81,A -85,B 0,C 180,E1 10207.912,E2 10207.912} C_VEL
LIN {X 0,Y 403.124,Z 526.81,A -85,B 0,C 180,E1 10214.464,E2 10214.464} C_VEL
LIN {X 0,Y 403.131,Z 526.81,A -85,B 0,C 180,E1 10220.315,E2 10220.315} C_VEL
LIN {X 0,Y 403.215,Z 526.81,A -85,B 0,C 180,E1 10225.713,E2 10225.713} C_VEL
LIN {X 0,Y 403.329,Z 526.81,A -85,B 0,C 180,E1 10230.784,E2 10230.784} C_VEL
LIN {X 0,Y 403.628,Z 526.81,A -85,B 0,C 180,E1 10237.963,E2 10237.963} C_VEL
LIN {X 0,Y 403.78,Z 526.81,A -85,B 0,C 180,E1 10244.777,E2 10244.777} C_VEL
LIN {X 0,Y 404.081,Z 526.81,A -85,B 0,C 180,E1 10251.512,E2 10251.512} C_VEL
LIN {X 0,Y 404.504,Z 526.81,A -85,B 0,C 180,E1 10257.848,E2 10257.848} C_VEL
LIN {X 0,Y 404.342,Z 526.81,A -85,B 0,C 180,E1 10264.288,E2 10264.288} C_VEL
LIN {X 0,Y 403.945,Z 526.81,A -85,B 0,C 180,E1 10270.794,E2 10270.794} C_VEL
LIN {X 0,Y 403.769,Z 526.81,A -85,B 0,C 180,E1 10277.449,E2 10277.449} C_VEL
LIN {X 0,Y 403.453,Z 526.81,A -85,B 0,C 180,E1 10284.373,E2 10284.373} C_VEL
LIN {X 0,Y 403.317,Z 526.81,A -85,B 0,C 180,E1 10291.697,E2 10291.697} C_VEL
LIN {X 0,Y 403.095,Z 526.81,A -85,B 0,C 180,E1 10297.936,E2 10297.936} C_VEL
LIN {X 0,Y 403.006,Z 526.81,A -85,B 0,C 180,E1 10304.461,E2 10304.461} C_VEL
LIN {X 0,Y 402.992,Z 526.81,A -85,B 0,C 180,E1 10310.312,E2 10310.312} C_VEL
LIN {X 0,Y 403.152,Z 526.81,A -85,B 0,C 180,E1 10315.719,E2 10315.719} C_VEL
LIN {X 0,Y 403.436,Z 526.81,A -85,B 0,C 180,E1 10320.05,E2 10320.05} C_VEL
LIN {X 0,Y 417.563,Z 573.757,A -85,B 0,C 180,E1 10321.719,E2 10321.719} C_VEL
LIN {X 0,Y 416.241,Z 610.153,A -85,B 0,C 180,E1 10322.731,E2 10322.731} C_VEL
LIN {X 0,Y 413.871,Z 641.992,A -85,B 0,C 180,E1 10324.402,E2 10324.402} C_VEL
LIN {X 0,Y 411.094,Z 672.982,A -85,B 0,C 180,E1 10326.93,E2 10326.93} C_VEL
LIN {X 0,Y 408.407,Z 700.804,A -85,B 0,C 180,E1 10330.233,E2 10330.233} C_VEL
LIN {X 0,Y 406.578,Z 723.532,A -85,B 0,C 180,E1 10334.065,E2 10334.065} C_VEL
LIN {X 0,Y 406.091,Z 731.704,A -85,B 0,C 180,E1 10335.844,E2 10335.844} C_VEL
LIN {X 0,Y 403.361,Z 737.856,A -85,B 0,C 180,E1 10337.442,E2 10337.442} C_VEL
LIN {X 0,Y 397.732,Z 745.366,A -85,B 0,C 180,E1 10339.956,E2 10339.956} C_VEL
LIN {X 0,Y 397.641,Z 746.134,A -85,B 0,C 180,E1 10340.254,E2 10340.254} C_VEL
LIN {X 0,Y 397.773,Z 754.876,A -85,B 0,C 180,E1 10344.545,E2 10344.545} C_VEL
LIN {X 0,Y 397.863,Z 758.162,A -85,B 0,C 180,E1 10347.824,E2 10347.824} C_VEL
LIN {X 0,Y 397.855,Z 758.003,A -85,B 0,C 180,E1 10352.186,E2 10352.186} C_VEL
LIN {X 0,Y 397.796,Z 752.816,A -85,B 0,C 180,E1 10356.562,E2 10356.562} C_VEL
LIN {X 0,Y 397.75,Z 742.21,A -85,B 0,C 180,E1 10360.977,E2 10360.977} C_VEL
LIN {X 0,Y 398.532,Z 725.588,A -85,B 0,C 180,E1 10365.428,E2 10365.428} C_VEL
LIN {X 0,Y 400.361,Z 703.038,A -85,B 0,C 180,E1 10369.602,E2 10369.602} C_VEL
LIN {X 0,Y 403.282,Z 675.695,A -85,B 0,C 180,E1 10373.191,E2 10373.191} C_VEL
LIN {X 0,Y 406.566,Z 645.703,A -85,B 0,C 180,E1 10375.955,E2 10375.955} C_VEL
LIN {X 0,Y 409.856,Z 611.892,A -85,B 0,C 180,E1 10378.011,E2 10378.011} C_VEL
LIN {X 0,Y 412.044,Z 576.567,A -85,B 0,C 180,E1 10379.216,E2 10379.216} C_VEL
LIN {X 0,Y 408.389,Z 558.844,A -85,B 0,C 180,E1 10379.958,E2 10379.958} C_VEL
LIN {X 0,Y 397.297,Z 531.986,A -85,B 0,C 180,E1 10381.75,E2 10381.75} C_VEL
LIN {X 0,Y 395.282,Z 526.81,A -85,B 0,C 180,E1 10382.233,E2 10382.233} C_VEL
LIN {X 0,Y 395.21,Z 526.81,A -85,B 0,C 180,E1 10387.811,E2 10387.811} C_VEL
LIN {X 0,Y 395.264,Z 526.81,A -85,B 0,C 180,E1 10393.597,E2 10393.597} C_VEL
LIN {X 0,Y 395.218,Z 526.81,A -85,B 0,C 180,E1 10400.021,E2 10400.021} C_VEL
LIN {X 0,Y 395.315,Z 526.81,A -85,B 0,C 180,E1 10407.584,E2 10407.584} C_VEL
LIN {X 0,Y 395.421,Z 526.81,A -85,B 0,C 180,E1 10412.656,E2 10412.656} C_VEL
LIN {X 0,Y 395.684,Z 527.456,A -85,B 0,C 180,E1 10418.383,E2 10418.383} C_VEL
LIN {X 0,Y 404.958,Z 553.565,A -85,B 0,C 180,E1 10420.615,E2 10420.615} C_VEL
LIN {X 0,Y 407.205,Z 570.75,A -85,B 0,C 180,E1 10422.053,E2 10422.053} C_VEL
LIN {X 0,Y 404.763,Z 596.722,A -85,B 0,C 180,E1 10424.55,E2 10424.55} C_VEL
LIN {X 0,Y 402.529,Z 616.686,A -85,B 0,C 180,E1 10427.476,E2 10427.476} C_VEL
LIN {X 0,Y 400.746,Z 631.329,A -85,B 0,C 180,E1 10430.767,E2 10430.767} C_VEL
LIN {X 0,Y 399.524,Z 641.092,A -85,B 0,C 180,E1 10434.571,E2 10434.571} C_VEL
LIN {X 0,Y 398.848,Z 644.512,A -85,B 0,C 180,E1 10437.831,E2 10437.831} C_VEL
LIN {X 0,Y 398.587,Z 644.408,A -85,B 0,C 180,E1 10440.007,E2 10440.007} C_VEL
LIN {X 0,Y 398.497,Z 639.778,A -85,B 0,C 180,E1 10443.819,E2 10443.819} C_VEL
LIN {X 0,Y 399.023,Z 628.913,A -85,B 0,C 180,E1 10447.638,E2 10447.638} C_VEL
LIN {X 0,Y 399.951,Z 613.473,A -85,B 0,C 180,E1 10450.917,E2 10450.917} C_VEL
LIN {X 0,Y 401.332,Z 592.013,A -85,B 0,C 180,E1 10453.922,E2 10453.922} C_VEL
LIN {X 0,Y 402.888,Z 566.365,A -85,B 0,C 180,E1 10456.271,E2 10456.271} C_VEL
LIN {X 0,Y 400.068,Z 546.371,A -85,B 0,C 180,E1 10457.63,E2 10457.63} C_VEL
LIN {X 0,Y 395.925,Z 526.81,A -85,B 0,C 180,E1 10458.686,E2 10458.686} C_VEL
LIN {X 0,Y 395.546,Z 526.81,A -85,B 0,C 180,E1 10464.907,E2 10464.907} C_VEL
LIN {X 0,Y 395.409,Z 526.81,A -85,B 0,C 180,E1 10469.86,E2 10469.86} C_VEL
LIN {X 0,Y 395.19,Z 526.81,A -85,B 0,C 180,E1 10477.813,E2 10477.813} C_VEL
LIN {X 0,Y 395.178,Z 526.81,A -85,B 0,C 180,E1 10483.608,E2 10483.608} C_VEL
LIN {X 0,Y 395.249,Z 526.81,A -85,B 0,C 180,E1 10490.015,E2 10490.015} C_VEL
LIN {X 0,Y 395.305,Z 526.81,A -85,B 0,C 180,E1 10497.567,E2 10497.567} C_VEL
LIN {X 0,Y 395.455,Z 526.81,A -85,B 0,C 180,E1 10502.643,E2 10502.643} C_VEL
LIN {X 0,Y 395.78,Z 526.81,A -85,B 0,C 180,E1 10509.856,E2 10509.856} C_VEL
LIN {X 0,Y 395.875,Z 526.81,A -85,B 0,C 180,E1 10516.728,E2 10516.728} C_VEL
LIN {X 0,Y 396.3,Z 526.81,A -85,B 0,C 180,E1 10523.413,E2 10523.413} C_VEL
LIN {X 0,Y 396.65,Z 526.81,A -85,B 0,C 180,E1 10529.995,E2 10529.995} C_VEL
LIN {X 0,Y 396.291,Z 526.81,A -85,B 0,C 180,E1 10536.576,E2 10536.576} C_VEL
LIN {X 0,Y 395.991,Z 526.81,A -85,B 0,C 180,E1 10543.257,E2 10543.257} C_VEL
LIN {X 0,Y 395.765,Z 526.81,A -85,B 0,C 180,E1 10550.134,E2 10550.134} C_VEL
LIN {X 0,Y 395.414,Z 526.81,A -85,B 0,C 180,E1 10557.348,E2 10557.348} C_VEL
LIN {X 0,Y 395.285,Z 526.81,A -85,B 0,C 180,E1 10562.569,E2 10562.569} C_VEL
LIN {X 0,Y 395.166,Z 526.81,A -85,B 0,C 180,E1 10569.971,E2 10569.971} C_VEL
LIN {X 0,Y 395.192,Z 526.81,A -85,B 0,C 180,E1 10576.706,E2 10576.706} C_VEL
LIN {X 0,Y 395.194,Z 526.81,A -85,B 0,C 180,E1 10583.558,E2 10583.558} C_VEL
LIN {X 0,Y 395.4,Z 526.81,A -85,B 0,C 180,E1 10590.14,E2 10590.14} C_VEL
LIN {X 0,Y 395.643,Z 526.81,A -85,B 0,C 180,E1 10597.494,E2 10597.494} C_VEL
LIN {X 0,Y 395.843,Z 526.81,A -85,B 0,C 180,E1 10604.464,E2 10604.464} C_VEL
LIN {X 0,Y 396.145,Z 526.81,A -85,B 0,C 180,E1 10611.508,E2 10611.508} C_VEL
LIN {X 0,Y 396.589,Z 526.81,A -85,B 0,C 180,E1 10617.805,E2 10617.805} C_VEL
LIN {X 0,Y 396.421,Z 526.81,A -85,B 0,C 180,E1 10624.374,E2 10624.374} C_VEL
LIN {X 0,Y 396.012,Z 526.81,A -85,B 0,C 180,E1 10631.013,E2 10631.013} C_VEL
